LIN {X 0,Y 488.521,Z 455.638,A -85,B 0,C 180,E1 -6694.13,E2 -6694.13} C_VEL
LIN {X 0,Y 488.662,Z 455.615,A -85,B 0,C 180,E1 -6696.351,E2 -6696.351} C_VEL
LIN {X 0,Y 488.705,Z 455.608,A -85,B 0,C 180,E1 -6699.254,E2 -6699.254} C_VEL
LIN {X 0,Y 488.728,Z 455.605,A -85,B 0,C 180,E1 -6701.602,E2 -6701.602} C_VEL
LIN {X 0,Y 488.717,Z 455.607,A -85,B 0,C 180,E1 -6704.802,E2 -6704.802} C_VEL
LIN {X 0,Y 488.696,Z 455.613,A -85,B 0,C 180,E1 -6707.475,E2 -6707.475} C_VEL
LIN {X 0,Y 488.738,Z 455.605,A -85,B 0,C 180,E1 -6709.677,E2 -6709.677} C_VEL
LIN {X 0,Y 488.684,Z 455.611,A -85,B 0,C 180,E1 -6712.841,E2 -6712.841} C_VEL
LIN {X 0,Y 488.736,Z 455.609,A -85,B 0,C 180,E1 -6715.887,E2 -6715.887} C_VEL
LIN {X 0,Y 488.697,Z 455.611,A -85,B 0,C 180,E1 -6718.82,E2 -6718.82} C_VEL
LIN {X 0,Y 488.713,Z 455.608,A -85,B 0,C 180,E1 -6720.348,E2 -6720.348} C_VEL
LIN {X 0,Y 488.06,Z 455.692,A -85,B 0,C 180,E1 -6721.037,E2 -6721.037} C_VEL
LIN {X 0,Y 485.216,Z 456.044,A -85,B 0,C 180,E1 -6722.155,E2 -6722.155} C_VEL
LIN {X 0,Y 482.806,Z 456.345,A -85,B 0,C 180,E1 -6723.056,E2 -6723.056} C_VEL
LIN {X 0,Y 481.776,Z 456.472,A -85,B 0,C 180,E1 -6723.752,E2 -6723.752} C_VEL
LIN {X 0,Y 481.694,Z 456.483,A -85,B 0,C 180,E1 -6723.987,E2 -6723.987} C_VEL
LIN {X 0,Y 481.679,Z 456.482,A -85,B 0,C 180,E1 -6726.812,E2 -6726.812} C_VEL
LIN {X 0,Y 481.701,Z 456.483,A -85,B 0,C 180,E1 -6729.503,E2 -6729.503} C_VEL
LIN {X 0,Y 481.698,Z 456.482,A -85,B 0,C 180,E1 -6732.158,E2 -6732.158} C_VEL
LIN {X 0,Y 481.749,Z 456.478,A -85,B 0,C 180,E1 -6734.776,E2 -6734.776} C_VEL
LIN {X 0,Y 481.757,Z 456.478,A -85,B 0,C 180,E1 -6738.215,E2 -6738.215} C_VEL
LIN {X 0,Y 481.768,Z 456.476,A -85,B 0,C 180,E1 -6741.612,E2 -6741.612} C_VEL
LIN {X 0,Y 481.821,Z 456.467,A -85,B 0,C 180,E1 -6744.14,E2 -6744.14} C_VEL
LIN {X 0,Y 481.933,Z 456.452,A -85,B 0,C 180,E1 -6747.493,E2 -6747.493} C_VEL
LIN {X 0,Y 481.892,Z 456.456,A -85,B 0,C 180,E1 -6750.836,E2 -6750.836} C_VEL
LIN {X 0,Y 481.933,Z 456.452,A -85,B 0,C 180,E1 -6752.507,E2 -6752.507} C_VEL
LIN {X 0,Y 481.804,Z 456.47,A -85,B 0,C 180,E1 -6755.861,E2 -6755.861} C_VEL
LIN {X 0,Y 481.746,Z 456.478,A -85,B 0,C 180,E1 -6758.389,E2 -6758.389} C_VEL
LIN {X 0,Y 481.757,Z 456.475,A -85,B 0,C 180,E1 -6761.785,E2 -6761.785} C_VEL
LIN {X 0,Y 481.749,Z 456.475,A -85,B 0,C 180,E1 -6765.224,E2 -6765.224} C_VEL
LIN {X 0,Y 481.718,Z 456.481,A -85,B 0,C 180,E1 -6768.722,E2 -6768.722} C_VEL
LIN {X 0,Y 481.651,Z 456.488,A -85,B 0,C 180,E1 -6771.395,E2 -6771.395} C_VEL
LIN {X 0,Y 481.667,Z 456.49,A -85,B 0,C 180,E1 -6774.114,E2 -6774.114} C_VEL
LIN {X 0,Y 481.752,Z 456.474,A -85,B 0,C 180,E1 -6777.139,E2 -6777.139} C_VEL
LIN {X 0,Y 481.684,Z 456.485,A -85,B 0,C 180,E1 -6779.741,E2 -6779.741} C_VEL
LIN {X 0,Y 481.677,Z 456.487,A -85,B 0,C 180,E1 -6782.674,E2 -6782.674} C_VEL
LIN {X 0,Y 481.647,Z 456.489,A -85,B 0,C 180,E1 -6785.709,E2 -6785.709} C_VEL
LIN {X 0,Y 481.675,Z 456.482,A -85,B 0,C 180,E1 -6788.859,E2 -6788.859} C_VEL
LIN {X 0,Y 481.657,Z 456.487,A -85,B 0,C 180,E1 -6791.913,E2 -6791.913} C_VEL
LIN {X 0,Y 481.664,Z 456.488,A -85,B 0,C 180,E1 -6794.457,E2 -6794.457} C_VEL
LIN {X 0,Y 481.658,Z 456.488,A -85,B 0,C 180,E1 -6797.84,E2 -6797.84} C_VEL
LIN {X 0,Y 481.684,Z 456.482,A -85,B 0,C 180,E1 -6800.651,E2 -6800.651} C_VEL
LIN {X 0,Y 481.626,Z 456.494,A -85,B 0,C 180,E1 -6803.377,E2 -6803.377} C_VEL
LIN {X 0,Y 481.493,Z 456.51,A -85,B 0,C 180,E1 -6806.312,E2 -6806.312} C_VEL
LIN {X 0,Y 481.114,Z 456.559,A -85,B 0,C 180,E1 -6809.251,E2 -6809.251} C_VEL
LIN {X 0,Y 480.986,Z 456.764,A -85,B 0,C 180,E1 -6810.211,E2 -6810.211} C_VEL
LIN {X 0,Y 481.053,Z 460.075,A -85,B 0,C 180,E1 -6813.07,E2 -6813.07} C_VEL
LIN {X 0,Y 480.958,Z 463.269,A -85,B 0,C 180,E1 -6815.848,E2 -6815.848} C_VEL
LIN {X 0,Y 480.961,Z 467.196,A -85,B 0,C 180,E1 -6819.26,E2 -6819.26} C_VEL
LIN {X 0,Y 480.903,Z 470.487,A -85,B 0,C 180,E1 -6822.127,E2 -6822.127} C_VEL
LIN {X 0,Y 480.927,Z 474.157,A -85,B 0,C 180,E1 -6825.22,E2 -6825.22} C_VEL
LIN {X 0,Y 483.363,Z 485.552,A -85,B 0,C 180,E1 -6825.63,E2 -6825.63} C_VEL
LIN {X 0,Y 483.879,Z 489.967,A -85,B 0,C 180,E1 -6825.812,E2 -6825.812} C_VEL
LIN {X 0,Y 483.545,Z 501.529,A -85,B 0,C 180,E1 -6826.338,E2 -6826.338} C_VEL
LIN {X 0,Y 483.189,Z 513.218,A -85,B 0,C 180,E1 -6827.039,E2 -6827.039} C_VEL
LIN {X 0,Y 482.8,Z 524.711,A -85,B 0,C 180,E1 -6827.921,E2 -6827.921} C_VEL
LIN {X 0,Y 482.34,Z 534.688,A -85,B 0,C 180,E1 -6828.868,E2 -6828.868} C_VEL
LIN {X 0,Y 481.958,Z 543.707,A -85,B 0,C 180,E1 -6829.922,E2 -6829.922} C_VEL
LIN {X 0,Y 481.613,Z 552.483,A -85,B 0,C 180,E1 -6831.186,E2 -6831.186} C_VEL
LIN {X 0,Y 481.294,Z 559.557,A -85,B 0,C 180,E1 -6832.448,E2 -6832.448} C_VEL
LIN {X 0,Y 481.172,Z 565.776,A -85,B 0,C 180,E1 -6833.869,E2 -6833.869} C_VEL
LIN {X 0,Y 481.008,Z 570.825,A -85,B 0,C 180,E1 -6835.39,E2 -6835.39} C_VEL
LIN {X 0,Y 480.913,Z 573.824,A -85,B 0,C 180,E1 -6836.649,E2 -6836.649} C_VEL
LIN {X 0,Y 480.926,Z 575.286,A -85,B 0,C 180,E1 -6837.487,E2 -6837.487} C_VEL
LIN {X 0,Y 480.76,Z 576.965,A -85,B 0,C 180,E1 -6839.162,E2 -6839.162} C_VEL
LIN {X 0,Y 480.745,Z 577.228,A -85,B 0,C 180,E1 -6840,E2 -6840} C_VEL
LIN {X 0,Y 480.76,Z 577.054,A -85,B 0,C 180,E1 -6840.837,E2 -6840.837} C_VEL
LIN {X 0,Y 480.928,Z 575.521,A -85,B 0,C 180,E1 -6842.512,E2 -6842.512} C_VEL
LIN {X 0,Y 480.922,Z 574.16,A -85,B 0,C 180,E1 -6843.351,E2 -6843.351} C_VEL
LIN {X 0,Y 481.007,Z 571.287,A -85,B 0,C 180,E1 -6844.609,E2 -6844.609} C_VEL
LIN {X 0,Y 481.174,Z 566.349,A -85,B 0,C 180,E1 -6846.141,E2 -6846.141} C_VEL
LIN {X 0,Y 481.337,Z 560.311,A -85,B 0,C 180,E1 -6847.551,E2 -6847.551} C_VEL
LIN {X 0,Y 481.621,Z 553.395,A -85,B 0,C 180,E1 -6848.813,E2 -6848.813} C_VEL
LIN {X 0,Y 481.942,Z 544.787,A -85,B 0,C 180,E1 -6850.078,E2 -6850.078} C_VEL
LIN {X 0,Y 482.343,Z 535.961,A -85,B 0,C 180,E1 -6851.131,E2 -6851.131} C_VEL
LIN {X 0,Y 482.771,Z 526.199,A -85,B 0,C 180,E1 -6852.079,E2 -6852.079} C_VEL
LIN {X 0,Y 483.125,Z 514.56,A -85,B 0,C 180,E1 -6852.99,E2 -6852.99} C_VEL
LIN {X 0,Y 483.53,Z 502.682,A -85,B 0,C 180,E1 -6853.715,E2 -6853.715} C_VEL
LIN {X 0,Y 483.91,Z 489.989,A -85,B 0,C 180,E1 -6854.294,E2 -6854.294} C_VEL
LIN {X 0,Y 482.628,Z 482.026,A -85,B 0,C 180,E1 -6854.618,E2 -6854.618} C_VEL
LIN {X 0,Y 481.021,Z 475.218,A -85,B 0,C 180,E1 -6854.868,E2 -6854.868} C_VEL
LIN {X 0,Y 481.048,Z 471.328,A -85,B 0,C 180,E1 -6858.261,E2 -6858.261} C_VEL
LIN {X 0,Y 480.998,Z 467.621,A -85,B 0,C 180,E1 -6861.425,E2 -6861.425} C_VEL
LIN {X 0,Y 481.043,Z 464.368,A -85,B 0,C 180,E1 -6864.147,E2 -6864.147} C_VEL
LIN {X 0,Y 481.084,Z 460.834,A -85,B 0,C 180,E1 -6866.984,E2 -6866.984} C_VEL
LIN {X 0,Y 481.016,Z 456.971,A -85,B 0,C 180,E1 -6869.786,E2 -6869.786} C_VEL
LIN {X 0,Y 481.124,Z 456.558,A -85,B 0,C 180,E1 -6870.748,E2 -6870.748} C_VEL
LIN {X 0,Y 481.507,Z 456.51,A -85,B 0,C 180,E1 -6873.699,E2 -6873.699} C_VEL
LIN {X 0,Y 481.624,Z 456.494,A -85,B 0,C 180,E1 -6876.747,E2 -6876.747} C_VEL
LIN {X 0,Y 481.679,Z 456.486,A -85,B 0,C 180,E1 -6879.94,E2 -6879.94} C_VEL
LIN {X 0,Y 481.669,Z 456.488,A -85,B 0,C 180,E1 -6883.297,E2 -6883.297} C_VEL
LIN {X 0,Y 481.661,Z 456.49,A -85,B 0,C 180,E1 -6885.641,E2 -6885.641} C_VEL
LIN {X 0,Y 481.659,Z 456.489,A -85,B 0,C 180,E1 -6888.958,E2 -6888.958} C_VEL
LIN {X 0,Y 481.719,Z 456.635,A -85,B 0,C 180,E1 -6889.998,E2 -6889.998} C_VEL
LIN {X 0,Y 483.121,Z 464.541,A -85,B 0,C 180,E1 -6893.385,E2 -6893.385} C_VEL
LIN {X 0,Y 483.304,Z 468.523,A -85,B 0,C 180,E1 -6894.987,E2 -6894.987} C_VEL
LIN {X 0,Y 482.858,Z 476.355,A -85,B 0,C 180,E1 -6897.987,E2 -6897.987} C_VEL
LIN {X 0,Y 482.423,Z 484.318,A -85,B 0,C 180,E1 -6900.937,E2 -6900.937} C_VEL
LIN {X 0,Y 482.124,Z 491.72,A -85,B 0,C 180,E1 -6903.602,E2 -6903.602} C_VEL
LIN {X 0,Y 481.857,Z 499.554,A -85,B 0,C 180,E1 -6906.354,E2 -6906.354} C_VEL
LIN {X 0,Y 481.566,Z 508.719,A -85,B 0,C 180,E1 -6909.497,E2 -6909.497} C_VEL
LIN {X 0,Y 481.343,Z 517.918,A -85,B 0,C 180,E1 -6912.583,E2 -6912.583} C_VEL
LIN {X 0,Y 481.207,Z 525.513,A -85,B 0,C 180,E1 -6915.083,E2 -6915.083} C_VEL
LIN {X 0,Y 483.109,Z 538.984,A -85,B 0,C 180,E1 -6915.494,E2 -6915.494} C_VEL
LIN {X 0,Y 483.716,Z 544.262,A -85,B 0,C 180,E1 -6915.7,E2 -6915.7} C_VEL
LIN {X 0,Y 483.348,Z 556.096,A -85,B 0,C 180,E1 -6916.226,E2 -6916.226} C_VEL
LIN {X 0,Y 482.981,Z 567.433,A -85,B 0,C 180,E1 -6916.89,E2 -6916.89} C_VEL
LIN {X 0,Y 482.477,Z 579.715,A -85,B 0,C 180,E1 -6917.809,E2 -6917.809} C_VEL
LIN {X 0,Y 482.083,Z 589.793,A -85,B 0,C 180,E1 -6918.756,E2 -6918.756} C_VEL
LIN {X 0,Y 481.628,Z 599.758,A -85,B 0,C 180,E1 -6919.915,E2 -6919.915} C_VEL
LIN {X 0,Y 481.333,Z 608.553,A -85,B 0,C 180,E1 -6921.181,E2 -6921.181} C_VEL
LIN {X 0,Y 481.107,Z 615.571,A -85,B 0,C 180,E1 -6922.445,E2 -6922.445} C_VEL
LIN {X 0,Y 480.938,Z 621.582,A -85,B 0,C 180,E1 -6923.809,E2 -6923.809} C_VEL
LIN {X 0,Y 480.905,Z 625.601,A -85,B 0,C 180,E1 -6924.97,E2 -6924.97} C_VEL
LIN {X 0,Y 480.858,Z 627.928,A -85,B 0,C 180,E1 -6925.809,E2 -6925.809} C_VEL
LIN {X 0,Y 480.894,Z 629.821,A -85,B 0,C 180,E1 -6926.649,E2 -6926.649} C_VEL
LIN {X 0,Y 480.869,Z 631.238,A -85,B 0,C 180,E1 -6927.487,E2 -6927.487} C_VEL
LIN {X 0,Y 480.824,Z 632.239,A -85,B 0,C 180,E1 -6928.325,E2 -6928.325} C_VEL
LIN {X 0,Y 480.742,Z 633.044,A -85,B 0,C 180,E1 -6930,E2 -6930} C_VEL
LIN {X 0,Y 480.76,Z 632.811,A -85,B 0,C 180,E1 -6930.838,E2 -6930.838} C_VEL
LIN {X 0,Y 480.825,Z 632.176,A -85,B 0,C 180,E1 -6931.675,E2 -6931.675} C_VEL
LIN {X 0,Y 480.881,Z 631.139,A -85,B 0,C 180,E1 -6932.513,E2 -6932.513} C_VEL
LIN {X 0,Y 480.894,Z 629.685,A -85,B 0,C 180,E1 -6933.351,E2 -6933.351} C_VEL
LIN {X 0,Y 480.853,Z 626.643,A -85,B 0,C 180,E1 -6934.611,E2 -6934.611} C_VEL
LIN {X 0,Y 480.953,Z 622.538,A -85,B 0,C 180,E1 -6935.871,E2 -6935.871} C_VEL
LIN {X 0,Y 481.108,Z 616.224,A -85,B 0,C 180,E1 -6937.344,E2 -6937.344} C_VEL
LIN {X 0,Y 481.303,Z 609.329,A -85,B 0,C 180,E1 -6938.608,E2 -6938.608} C_VEL
LIN {X 0,Y 481.537,Z 600.775,A -85,B 0,C 180,E1 -6939.875,E2 -6939.875} C_VEL
LIN {X 0,Y 481.902,Z 591.982,A -85,B 0,C 180,E1 -6940.929,E2 -6940.929} C_VEL
LIN {X 0,Y 482.32,Z 581.32,A -85,B 0,C 180,E1 -6941.972,E2 -6941.972} C_VEL
LIN {X 0,Y 482.723,Z 570.803,A -85,B 0,C 180,E1 -6942.807,E2 -6942.807} C_VEL
LIN {X 0,Y 483.189,Z 558.755,A -85,B 0,C 180,E1 -6943.564,E2 -6943.564} C_VEL
LIN {X 0,Y 483.574,Z 545.487,A -85,B 0,C 180,E1 -6944.197,E2 -6944.197} C_VEL
LIN {X 0,Y 483.219,Z 540.19,A -85,B 0,C 180,E1 -6944.409,E2 -6944.409} C_VEL
LIN {X 0,Y 481.464,Z 526.61,A -85,B 0,C 180,E1 -6944.854,E2 -6944.854} C_VEL
LIN {X 0,Y 481.177,Z 524.25,A -85,B 0,C 180,E1 -6944.918,E2 -6944.918} C_VEL
LIN {X 0,Y 481.251,Z 515.065,A -85,B 0,C 180,E1 -6947.859,E2 -6947.859} C_VEL
LIN {X 0,Y 481.488,Z 505.759,A -85,B 0,C 180,E1 -6950.905,E2 -6950.905} C_VEL
LIN {X 0,Y 481.688,Z 496.306,A -85,B 0,C 180,E1 -6954.113,E2 -6954.113} C_VEL
LIN {X 0,Y 482.022,Z 487.666,A -85,B 0,C 180,E1 -6957.202,E2 -6957.202} C_VEL
LIN {X 0,Y 482.372,Z 479.925,A -85,B 0,C 180,E1 -6960.176,E2 -6960.176} C_VEL
LIN {X 0,Y 482.874,Z 473.051,A -85,B 0,C 180,E1 -6963.079,E2 -6963.079} C_VEL
LIN {X 0,Y 483.32,Z 467.859,A -85,B 0,C 180,E1 -6965.566,E2 -6965.566} C_VEL
LIN {X 0,Y 483.222,Z 465.5,A -85,B 0,C 180,E1 -6966.877,E2 -6966.877} C_VEL
LIN {X 0,Y 482.592,Z 461.645,A -85,B 0,C 180,E1 -6969.48,E2 -6969.48} C_VEL
LIN {X 0,Y 482.074,Z 458.808,A -85,B 0,C 180,E1 -6972.115,E2 -6972.115} C_VEL
LIN {X 0,Y 481.786,Z 457.245,A -85,B 0,C 180,E1 -6974.443,E2 -6974.443} C_VEL
LIN {X 0,Y 481.673,Z 456.489,A -85,B 0,C 180,E1 -6976.848,E2 -6976.848} C_VEL
LIN {X 0,Y 481.679,Z 456.602,A -85,B 0,C 180,E1 -6980.06,E2 -6980.06} C_VEL
LIN {X 0,Y 481.773,Z 457.262,A -85,B 0,C 180,E1 -6982.216,E2 -6982.216} C_VEL
LIN {X 0,Y 481.851,Z 458.489,A -85,B 0,C 180,E1 -6984.764,E2 -6984.764} C_VEL
LIN {X 0,Y 481.721,Z 460.097,A -85,B 0,C 180,E1 -6987.33,E2 -6987.33} C_VEL
LIN {X 0,Y 481.564,Z 462.204,A -85,B 0,C 180,E1 -6990.251,E2 -6990.251} C_VEL
LIN {X 0,Y 481.44,Z 464.478,A -85,B 0,C 180,E1 -6993.094,E2 -6993.094} C_VEL
LIN {X 0,Y 481.289,Z 466.84,A -85,B 0,C 180,E1 -6995.866,E2 -6995.866} C_VEL
LIN {X 0,Y 481.221,Z 470.102,A -85,B 0,C 180,E1 -6999.482,E2 -6999.482} C_VEL
LIN {X 0,Y 481.133,Z 472.621,A -85,B 0,C 180,E1 -7002.137,E2 -7002.137} C_VEL
LIN {X 0,Y 481.11,Z 475.839,A -85,B 0,C 180,E1 -7005.23,E2 -7005.23} C_VEL
LIN {X 0,Y 483.747,Z 487.707,A -85,B 0,C 180,E1 -7005.684,E2 -7005.684} C_VEL
LIN {X 0,Y 483.728,Z 499.221,A -85,B 0,C 180,E1 -7006.183,E2 -7006.183} C_VEL
LIN {X 0,Y 483.295,Z 511.887,A -85,B 0,C 180,E1 -7006.901,E2 -7006.901} C_VEL
LIN {X 0,Y 482.929,Z 522.885,A -85,B 0,C 180,E1 -7007.712,E2 -7007.712} C_VEL
LIN {X 0,Y 482.459,Z 533.264,A -85,B 0,C 180,E1 -7008.659,E2 -7008.659} C_VEL
LIN {X 0,Y 482.094,Z 542.637,A -85,B 0,C 180,E1 -7009.713,E2 -7009.713} C_VEL
LIN {X 0,Y 481.725,Z 551.652,A -85,B 0,C 180,E1 -7010.977,E2 -7010.977} C_VEL
LIN {X 0,Y 481.397,Z 558.919,A -85,B 0,C 180,E1 -7012.239,E2 -7012.239} C_VEL
LIN {X 0,Y 481.213,Z 565.03,A -85,B 0,C 180,E1 -7013.575,E2 -7013.575} C_VEL
LIN {X 0,Y 480.932,Z 569.918,A -85,B 0,C 180,E1 -7014.97,E2 -7014.97} C_VEL
LIN {X 0,Y 481.044,Z 572.203,A -85,B 0,C 180,E1 -7015.811,E2 -7015.811} C_VEL
LIN {X 0,Y 480.922,Z 574.074,A -85,B 0,C 180,E1 -7016.649,E2 -7016.649} C_VEL
LIN {X 0,Y 480.928,Z 575.488,A -85,B 0,C 180,E1 -7017.488,E2 -7017.488} C_VEL
LIN {X 0,Y 480.76,Z 577.088,A -85,B 0,C 180,E1 -7019.163,E2 -7019.163} C_VEL
LIN {X 0,Y 480.744,Z 577.307,A -85,B 0,C 180,E1 -7020,E2 -7020} C_VEL
LIN {X 0,Y 480.76,Z 577.099,A -85,B 0,C 180,E1 -7020.838,E2 -7020.838} C_VEL
LIN {X 0,Y 480.926,Z 575.483,A -85,B 0,C 180,E1 -7022.513,E2 -7022.513} C_VEL
LIN {X 0,Y 480.913,Z 574.091,A -85,B 0,C 180,E1 -7023.351,E2 -7023.351} C_VEL
LIN {X 0,Y 481.003,Z 571.16,A -85,B 0,C 180,E1 -7024.61,E2 -7024.61} C_VEL
LIN {X 0,Y 481.182,Z 566.177,A -85,B 0,C 180,E1 -7026.14,E2 -7026.14} C_VEL
LIN {X 0,Y 481.301,Z 560.075,A -85,B 0,C 180,E1 -7027.552,E2 -7027.552} C_VEL
LIN {X 0,Y 481.599,Z 553.167,A -85,B 0,C 180,E1 -7028.814,E2 -7028.814} C_VEL
LIN {X 0,Y 481.939,Z 544.51,A -85,B 0,C 180,E1 -7030.079,E2 -7030.079} C_VEL
LIN {X 0,Y 482.304,Z 535.641,A -85,B 0,C 180,E1 -7031.133,E2 -7031.133} C_VEL
LIN {X 0,Y 482.769,Z 525.91,A -85,B 0,C 180,E1 -7032.08,E2 -7032.08} C_VEL
LIN {X 0,Y 483.06,Z 515.699,A -85,B 0,C 180,E1 -7032.895,E2 -7032.895} C_VEL
LIN {X 0,Y 483.492,Z 503.394,A -85,B 0,C 180,E1 -7033.663,E2 -7033.663} C_VEL
LIN {X 0,Y 483.857,Z 491.187,A -85,B 0,C 180,E1 -7034.242,E2 -7034.242} C_VEL
LIN {X 0,Y 483.271,Z 484.851,A -85,B 0,C 180,E1 -7034.502,E2 -7034.502} C_VEL
LIN {X 0,Y 480.957,Z 474.164,A -85,B 0,C 180,E1 -7034.898,E2 -7034.898} C_VEL
LIN {X 0,Y 480.962,Z 470.439,A -85,B 0,C 180,E1 -7038.23,E2 -7038.23} C_VEL
LIN {X 0,Y 480.953,Z 466.935,A -85,B 0,C 180,E1 -7041.427,E2 -7041.427} C_VEL
LIN {X 0,Y 480.987,Z 463.983,A -85,B 0,C 180,E1 -7044.15,E2 -7044.15} C_VEL
LIN {X 0,Y 481.089,Z 460.952,A -85,B 0,C 180,E1 -7046.985,E2 -7046.985} C_VEL
LIN {X 0,Y 481.117,Z 457.981,A -85,B 0,C 180,E1 -7049.78,E2 -7049.78} C_VEL
LIN {X 0,Y 481.128,Z 456.962,A -85,B 0,C 180,E1 -7050.748,E2 -7050.748} C_VEL
LIN {X 0,Y 481.22,Z 456.546,A -85,B 0,C 180,E1 -7052.106,E2 -7052.106} C_VEL
LIN {X 0,Y 481.573,Z 456.499,A -85,B 0,C 180,E1 -7055.189,E2 -7055.189} C_VEL
LIN {X 0,Y 481.654,Z 456.487,A -85,B 0,C 180,E1 -7058.007,E2 -7058.007} C_VEL
LIN {X 0,Y 481.667,Z 456.484,A -85,B 0,C 180,E1 -7061.041,E2 -7061.041} C_VEL
LIN {X 0,Y 481.664,Z 456.487,A -85,B 0,C 180,E1 -7064.36,E2 -7064.36} C_VEL
LIN {X 0,Y 481.637,Z 456.491,A -85,B 0,C 180,E1 -7066.853,E2 -7066.853} C_VEL
LIN {X 0,Y 481.681,Z 456.484,A -85,B 0,C 180,E1 -7070.06,E2 -7070.06} C_VEL
LIN {X 0,Y 481.63,Z 456.488,A -85,B 0,C 180,E1 -7073.253,E2 -7073.253} C_VEL
LIN {X 0,Y 481.715,Z 456.48,A -85,B 0,C 180,E1 -7076.33,E2 -7076.33} C_VEL
LIN {X 0,Y 481.656,Z 456.49,A -85,B 0,C 180,E1 -7079.417,E2 -7079.417} C_VEL
LIN {X 0,Y 481.705,Z 456.482,A -85,B 0,C 180,E1 -7082.168,E2 -7082.168} C_VEL
LIN {X 0,Y 481.694,Z 456.483,A -85,B 0,C 180,E1 -7083.987,E2 -7083.987} C_VEL
LIN {X 0,Y 481.031,Z 456.569,A -85,B 0,C 180,E1 -7084.685,E2 -7084.685} C_VEL
LIN {X 0,Y 478.163,Z 456.926,A -85,B 0,C 180,E1 -7085.819,E2 -7085.819} C_VEL
LIN {X 0,Y 475.729,Z 457.226,A -85,B 0,C 180,E1 -7086.732,E2 -7086.732} C_VEL
LIN {X 0,Y 474.677,Z 457.356,A -85,B 0,C 180,E1 -7087.438,E2 -7087.438} C_VEL
LIN {X 0,Y 474.588,Z 457.366,A -85,B 0,C 180,E1 -7087.677,E2 -7087.677} C_VEL
LIN {X 0,Y 474.66,Z 457.36,A -85,B 0,C 180,E1 -7090.09,E2 -7090.09} C_VEL
LIN {X 0,Y 474.645,Z 457.363,A -85,B 0,C 180,E1 -7092.774,E2 -7092.774} C_VEL
LIN {X 0,Y 474.654,Z 457.359,A -85,B 0,C 180,E1 -7095.421,E2 -7095.421} C_VEL
LIN {X 0,Y 474.711,Z 457.356,A -85,B 0,C 180,E1 -7098.038,E2 -7098.038} C_VEL
LIN {X 0,Y 474.733,Z 457.351,A -85,B 0,C 180,E1 -7101.487,E2 -7101.487} C_VEL
LIN {X 0,Y 474.784,Z 457.343,A -85,B 0,C 180,E1 -7104.052,E2 -7104.052} C_VEL
LIN {X 0,Y 474.899,Z 457.329,A -85,B 0,C 180,E1 -7107.455,E2 -7107.455} C_VEL
LIN {X 0,Y 474.918,Z 457.329,A -85,B 0,C 180,E1 -7110,E2 -7110} C_VEL
LIN {X 0,Y 474.899,Z 457.328,A -85,B 0,C 180,E1 -7112.545,E2 -7112.545} C_VEL
LIN {X 0,Y 474.765,Z 457.346,A -85,B 0,C 180,E1 -7115.948,E2 -7115.948} C_VEL
LIN {X 0,Y 474.717,Z 457.355,A -85,B 0,C 180,E1 -7118.514,E2 -7118.514} C_VEL
LIN {X 0,Y 474.711,Z 457.355,A -85,B 0,C 180,E1 -7121.962,E2 -7121.962} C_VEL
LIN {X 0,Y 474.706,Z 457.354,A -85,B 0,C 180,E1 -7125.456,E2 -7125.456} C_VEL
LIN {X 0,Y 474.67,Z 457.359,A -85,B 0,C 180,E1 -7129.01,E2 -7129.01} C_VEL
LIN {X 0,Y 474.594,Z 457.367,A -85,B 0,C 180,E1 -7131.729,E2 -7131.729} C_VEL
LIN {X 0,Y 474.646,Z 457.361,A -85,B 0,C 180,E1 -7134.494,E2 -7134.494} C_VEL
LIN {X 0,Y 474.686,Z 457.355,A -85,B 0,C 180,E1 -7137.334,E2 -7137.334} C_VEL
LIN {X 0,Y 474.61,Z 457.365,A -85,B 0,C 180,E1 -7140.23,E2 -7140.23} C_VEL
LIN {X 0,Y 474.648,Z 457.362,A -85,B 0,C 180,E1 -7143.22,E2 -7143.22} C_VEL
LIN {X 0,Y 474.597,Z 457.368,A -85,B 0,C 180,E1 -7146.323,E2 -7146.323} C_VEL
LIN {X 0,Y 474.632,Z 457.366,A -85,B 0,C 180,E1 -7149.647,E2 -7149.647} C_VEL
LIN {X 0,Y 474.619,Z 457.365,A -85,B 0,C 180,E1 -7152.934,E2 -7152.934} C_VEL
LIN {X 0,Y 474.62,Z 457.364,A -85,B 0,C 180,E1 -7155.896,E2 -7155.896} C_VEL
LIN {X 0,Y 474.637,Z 457.361,A -85,B 0,C 180,E1 -7159.04,E2 -7159.04} C_VEL
LIN {X 0,Y 474.614,Z 457.369,A -85,B 0,C 180,E1 -7161.704,E2 -7161.704} C_VEL
LIN {X 0,Y 474.56,Z 457.372,A -85,B 0,C 180,E1 -7164.72,E2 -7164.72} C_VEL
LIN {X 0,Y 474.296,Z 457.408,A -85,B 0,C 180,E1 -7167.761,E2 -7167.761} C_VEL
LIN {X 0,Y 473.993,Z 457.446,A -85,B 0,C 180,E1 -7169.726,E2 -7169.726} C_VEL
LIN {X 0,Y 473.921,Z 458.298,A -85,B 0,C 180,E1 -7171.038,E2 -7171.038} C_VEL
LIN {X 0,Y 473.947,Z 461.235,A -85,B 0,C 180,E1 -7173.585,E2 -7173.585} C_VEL
LIN {X 0,Y 473.881,Z 465.014,A -85,B 0,C 180,E1 -7176.854,E2 -7176.854} C_VEL
LIN {X 0,Y 473.842,Z 468.655,A -85,B 0,C 180,E1 -7180.054,E2 -7180.054} C_VEL
LIN {X 0,Y 473.8,Z 471.746,A -85,B 0,C 180,E1 -7182.742,E2 -7182.742} C_VEL
LIN {X 0,Y 473.825,Z 474.334,A -85,B 0,C 180,E1 -7184.991,E2 -7184.991} C_VEL
LIN {X 0,Y 476.597,Z 487.342,A -85,B 0,C 180,E1 -7185.482,E2 -7185.482} C_VEL
LIN {X 0,Y 476.931,Z 492.727,A -85,B 0,C 180,E1 -7185.71,E2 -7185.71} C_VEL
LIN {X 0,Y 476.508,Z 505.492,A -85,B 0,C 180,E1 -7186.35,E2 -7186.35} C_VEL
LIN {X 0,Y 476.154,Z 516.762,A -85,B 0,C 180,E1 -7187.087,E2 -7187.087} C_VEL
LIN {X 0,Y 475.767,Z 527.332,A -85,B 0,C 180,E1 -7187.956,E2 -7187.956} C_VEL
LIN {X 0,Y 475.222,Z 536.85,A -85,B 0,C 180,E1 -7188.915,E2 -7188.915} C_VEL
LIN {X 0,Y 474.888,Z 545.56,A -85,B 0,C 180,E1 -7189.986,E2 -7189.986} C_VEL
LIN {X 0,Y 474.52,Z 554.085,A -85,B 0,C 180,E1 -7191.268,E2 -7191.268} C_VEL
LIN {X 0,Y 474.247,Z 560.877,A -85,B 0,C 180,E1 -7192.549,E2 -7192.549} C_VEL
LIN {X 0,Y 474.087,Z 567.112,A -85,B 0,C 180,E1 -7194.043,E2 -7194.043} C_VEL
LIN {X 0,Y 473.926,Z 571.183,A -85,B 0,C 180,E1 -7195.321,E2 -7195.321} C_VEL
LIN {X 0,Y 473.848,Z 574.196,A -85,B 0,C 180,E1 -7196.599,E2 -7196.599} C_VEL
LIN {X 0,Y 473.866,Z 575.667,A -85,B 0,C 180,E1 -7197.45,E2 -7197.45} C_VEL
LIN {X 0,Y 473.689,Z 577.36,A -85,B 0,C 180,E1 -7199.15,E2 -7199.15} C_VEL
LIN {X 0,Y 473.672,Z 577.626,A -85,B 0,C 180,E1 -7200,E2 -7200} C_VEL
LIN {X 0,Y 473.689,Z 577.454,A -85,B 0,C 180,E1 -7200.85,E2 -7200.85} C_VEL
LIN {X 0,Y 473.868,Z 575.922,A -85,B 0,C 180,E1 -7202.55,E2 -7202.55} C_VEL
LIN {X 0,Y 473.856,Z 574.556,A -85,B 0,C 180,E1 -7203.401,E2 -7203.401} C_VEL
LIN {X 0,Y 473.944,Z 571.68,A -85,B 0,C 180,E1 -7204.678,E2 -7204.678} C_VEL
LIN {X 0,Y 474.085,Z 567.755,A -85,B 0,C 180,E1 -7205.956,E2 -7205.956} C_VEL
LIN {X 0,Y 474.218,Z 562.662,A -85,B 0,C 180,E1 -7207.237,E2 -7207.237} C_VEL
LIN {X 0,Y 474.498,Z 556.237,A -85,B 0,C 180,E1 -7208.518,E2 -7208.518} C_VEL
LIN {X 0,Y 474.817,Z 548.257,A -85,B 0,C 180,E1 -7209.8,E2 -7209.8} C_VEL
LIN {X 0,Y 475.204,Z 540.075,A -85,B 0,C 180,E1 -7210.869,E2 -7210.869} C_VEL
LIN {X 0,Y 475.69,Z 529.99,A -85,B 0,C 180,E1 -7211.937,E2 -7211.937} C_VEL
LIN {X 0,Y 476.075,Z 520.102,A -85,B 0,C 180,E1 -7212.793,E2 -7212.793} C_VEL
LIN {X 0,Y 476.455,Z 509.323,A -85,B 0,C 180,E1 -7213.549,E2 -7213.549} C_VEL
LIN {X 0,Y 476.9,Z 497.691,A -85,B 0,C 180,E1 -7214.182,E2 -7214.182} C_VEL
LIN {X 0,Y 476.924,Z 489.024,A -85,B 0,C 180,E1 -7214.561,E2 -7214.561} C_VEL
LIN {X 0,Y 474.354,Z 477.52,A -85,B 0,C 180,E1 -7215.032,E2 -7215.032} C_VEL
LIN {X 0,Y 473.95,Z 475.706,A -85,B 0,C 180,E1 -7215.102,E2 -7215.102} C_VEL
LIN {X 0,Y 473.979,Z 471.927,A -85,B 0,C 180,E1 -7218.382,E2 -7218.382} C_VEL
LIN {X 0,Y 473.934,Z 467.966,A -85,B 0,C 180,E1 -7221.76,E2 -7221.76} C_VEL
LIN {X 0,Y 473.983,Z 464.657,A -85,B 0,C 180,E1 -7224.53,E2 -7224.53} C_VEL
LIN {X 0,Y 474.003,Z 461.036,A -85,B 0,C 180,E1 -7227.363,E2 -7227.363} C_VEL
LIN {X 0,Y 474.009,Z 457.445,A -85,B 0,C 180,E1 -7230.272,E2 -7230.272} C_VEL
LIN {X 0,Y 474.391,Z 457.397,A -85,B 0,C 180,E1 -7233.24,E2 -7233.24} C_VEL
LIN {X 0,Y 474.566,Z 457.373,A -85,B 0,C 180,E1 -7235.46,E2 -7235.46} C_VEL
LIN {X 0,Y 474.613,Z 457.367,A -85,B 0,C 180,E1 -7238.457,E2 -7238.457} C_VEL
LIN {X 0,Y 474.634,Z 457.365,A -85,B 0,C 180,E1 -7240.96,E2 -7240.96} C_VEL
LIN {X 0,Y 474.618,Z 457.366,A -85,B 0,C 180,E1 -7244.104,E2 -7244.104} C_VEL
LIN {X 0,Y 474.617,Z 457.367,A -85,B 0,C 180,E1 -7247.066,E2 -7247.066} C_VEL
LIN {X 0,Y 474.671,Z 457.504,A -85,B 0,C 180,E1 -7249.738,E2 -7249.738} C_VEL
LIN {X 0,Y 475.936,Z 464.709,A -85,B 0,C 180,E1 -7252.883,E2 -7252.883} C_VEL
LIN {X 0,Y 476.32,Z 467.971,A -85,B 0,C 180,E1 -7254.244,E2 -7254.244} C_VEL
LIN {X 0,Y 476.008,Z 474.682,A -85,B 0,C 180,E1 -7256.887,E2 -7256.887} C_VEL
LIN {X 0,Y 475.595,Z 482.436,A -85,B 0,C 180,E1 -7259.839,E2 -7259.839} C_VEL
LIN {X 0,Y 475.216,Z 490.209,A -85,B 0,C 180,E1 -7262.712,E2 -7262.712} C_VEL
LIN {X 0,Y 474.836,Z 499.32,A -85,B 0,C 180,E1 -7265.982,E2 -7265.982} C_VEL
LIN {X 0,Y 474.49,Z 508.457,A -85,B 0,C 180,E1 -7269.177,E2 -7269.177} C_VEL
LIN {X 0,Y 474.3,Z 516.311,A -85,B 0,C 180,E1 -7271.87,E2 -7271.87} C_VEL
LIN {X 0,Y 474.166,Z 525.158,A -85,B 0,C 180,E1 -7274.857,E2 -7274.857} C_VEL
LIN {X 0,Y 476.178,Z 539.625,A -85,B 0,C 180,E1 -7275.319,E2 -7275.319} C_VEL
LIN {X 0,Y 476.792,Z 545.085,A -85,B 0,C 180,E1 -7275.542,E2 -7275.542} C_VEL
LIN {X 0,Y 476.357,Z 557.52,A -85,B 0,C 180,E1 -7276.128,E2 -7276.128} C_VEL
LIN {X 0,Y 475.918,Z 569.57,A -85,B 0,C 180,E1 -7276.877,E2 -7276.877} C_VEL
LIN {X 0,Y 475.419,Z 580.793,A -85,B 0,C 180,E1 -7277.765,E2 -7277.765} C_VEL
LIN {X 0,Y 475.031,Z 590.292,A -85,B 0,C 180,E1 -7278.695,E2 -7278.695} C_VEL
LIN {X 0,Y 474.593,Z 599.29,A -85,B 0,C 180,E1 -7279.764,E2 -7279.764} C_VEL
LIN {X 0,Y 474.272,Z 608.103,A -85,B 0,C 180,E1 -7281.049,E2 -7281.049} C_VEL
LIN {X 0,Y 474.038,Z 615.137,A -85,B 0,C 180,E1 -7282.332,E2 -7282.332} C_VEL
LIN {X 0,Y 473.88,Z 620.512,A -85,B 0,C 180,E1 -7283.547,E2 -7283.547} C_VEL
LIN {X 0,Y 473.839,Z 625.188,A -85,B 0,C 180,E1 -7284.894,E2 -7284.894} C_VEL
LIN {X 0,Y 473.76,Z 627.516,A -85,B 0,C 180,E1 -7285.746,E2 -7285.746} C_VEL
LIN {X 0,Y 473.82,Z 629.414,A -85,B 0,C 180,E1 -7286.599,E2 -7286.599} C_VEL
LIN {X 0,Y 473.783,Z 630.833,A -85,B 0,C 180,E1 -7287.449,E2 -7287.449} C_VEL
LIN {X 0,Y 473.758,Z 631.834,A -85,B 0,C 180,E1 -7288.3,E2 -7288.3} C_VEL
LIN {X 0,Y 473.688,Z 632.434,A -85,B 0,C 180,E1 -7289.15,E2 -7289.15} C_VEL
LIN {X 0,Y 473.669,Z 632.636,A -85,B 0,C 180,E1 -7290,E2 -7290} C_VEL
LIN {X 0,Y 473.688,Z 632.399,A -85,B 0,C 180,E1 -7290.85,E2 -7290.85} C_VEL
LIN {X 0,Y 473.758,Z 631.756,A -85,B 0,C 180,E1 -7291.7,E2 -7291.7} C_VEL
LIN {X 0,Y 473.793,Z 630.71,A -85,B 0,C 180,E1 -7292.551,E2 -7292.551} C_VEL
LIN {X 0,Y 473.821,Z 629.249,A -85,B 0,C 180,E1 -7293.401,E2 -7293.401} C_VEL
LIN {X 0,Y 473.775,Z 626.189,A -85,B 0,C 180,E1 -7294.68,E2 -7294.68} C_VEL
LIN {X 0,Y 473.859,Z 622.061,A -85,B 0,C 180,E1 -7295.959,E2 -7295.959} C_VEL
LIN {X 0,Y 474.017,Z 615.71,A -85,B 0,C 180,E1 -7297.454,E2 -7297.454} C_VEL
LIN {X 0,Y 474.213,Z 608.786,A -85,B 0,C 180,E1 -7298.738,E2 -7298.738} C_VEL
LIN {X 0,Y 474.495,Z 600.204,A -85,B 0,C 180,E1 -7300.023,E2 -7300.023} C_VEL
LIN {X 0,Y 474.897,Z 591.382,A -85,B 0,C 180,E1 -7301.092,E2 -7301.092} C_VEL
LIN {X 0,Y 475.329,Z 580.969,A -85,B 0,C 180,E1 -7302.126,E2 -7302.126} C_VEL
LIN {X 0,Y 475.791,Z 569.875,A -85,B 0,C 180,E1 -7303.018,E2 -7303.018} C_VEL
LIN {X 0,Y 476.238,Z 558.098,A -85,B 0,C 180,E1 -7303.766,E2 -7303.766} C_VEL
LIN {X 0,Y 476.671,Z 544.885,A -85,B 0,C 180,E1 -7304.407,E2 -7304.407} C_VEL
LIN {X 0,Y 475.105,Z 531.598,A -85,B 0,C 180,E1 -7304.921,E2 -7304.921} C_VEL
LIN {X 0,Y 474.114,Z 523.769,A -85,B 0,C 180,E1 -7305.145,E2 -7305.145} C_VEL
LIN {X 0,Y 474.241,Z 513.587,A -85,B 0,C 180,E1 -7308.477,E2 -7308.477} C_VEL
LIN {X 0,Y 474.465,Z 503.913,A -85,B 0,C 180,E1 -7311.735,E2 -7311.735} C_VEL
LIN {X 0,Y 474.736,Z 494.736,A -85,B 0,C 180,E1 -7314.956,E2 -7314.956} C_VEL
LIN {X 0,Y 475.041,Z 487.111,A -85,B 0,C 180,E1 -7317.786,E2 -7317.786} C_VEL
LIN {X 0,Y 475.545,Z 478.74,A -85,B 0,C 180,E1 -7321.149,E2 -7321.149} C_VEL
LIN {X 0,Y 476.132,Z 471.877,A -85,B 0,C 180,E1 -7324.249,E2 -7324.249} C_VEL
LIN {X 0,Y 476.319,Z 468.198,A -85,B 0,C 180,E1 -7326.171,E2 -7326.171} C_VEL
LIN {X 0,Y 475.912,Z 464.512,A -85,B 0,C 180,E1 -7328.494,E2 -7328.494} C_VEL
LIN {X 0,Y 475.366,Z 461.397,A -85,B 0,C 180,E1 -7331.061,E2 -7331.061} C_VEL
LIN {X 0,Y 474.94,Z 459.349,A -85,B 0,C 180,E1 -7333.524,E2 -7333.524} C_VEL
LIN {X 0,Y 474.745,Z 458.223,A -85,B 0,C 180,E1 -7335.911,E2 -7335.911} C_VEL
LIN {X 0,Y 474.711,Z 457.857,A -85,B 0,C 180,E1 -7338.224,E2 -7338.224} C_VEL
LIN {X 0,Y 474.718,Z 458.081,A -85,B 0,C 180,E1 -7340.461,E2 -7340.461} C_VEL
LIN {X 0,Y 474.805,Z 458.912,A -85,B 0,C 180,E1 -7343.064,E2 -7343.064} C_VEL
LIN {X 0,Y 474.789,Z 460.268,A -85,B 0,C 180,E1 -7345.772,E2 -7345.772} C_VEL
LIN {X 0,Y 474.628,Z 462.195,A -85,B 0,C 180,E1 -7348.785,E2 -7348.785} C_VEL
LIN {X 0,Y 474.456,Z 464.361,A -85,B 0,C 180,E1 -7351.705,E2 -7351.705} C_VEL
LIN {X 0,Y 474.315,Z 466.748,A -85,B 0,C 180,E1 -7354.669,E2 -7354.669} C_VEL
LIN {X 0,Y 474.176,Z 469.041,A -85,B 0,C 180,E1 -7357.334,E2 -7357.334} C_VEL
LIN {X 0,Y 474.091,Z 471.502,A -85,B 0,C 180,E1 -7360.065,E2 -7360.065} C_VEL
LIN {X 0,Y 474.043,Z 474.028,A -85,B 0,C 180,E1 -7362.752,E2 -7362.752} C_VEL
LIN {X 0,Y 474.039,Z 476.2,A -85,B 0,C 180,E1 -7364.985,E2 -7364.985} C_VEL
LIN {X 0,Y 476.869,Z 488.579,A -85,B 0,C 180,E1 -7365.49,E2 -7365.49} C_VEL
LIN {X 0,Y 476.863,Z 499.583,A -85,B 0,C 180,E1 -7365.98,E2 -7365.98} C_VEL
LIN {X 0,Y 476.481,Z 511.092,A -85,B 0,C 180,E1 -7366.634,E2 -7366.634} C_VEL
LIN {X 0,Y 476.058,Z 521.991,A -85,B 0,C 180,E1 -7367.423,E2 -7367.423} C_VEL
LIN {X 0,Y 475.575,Z 532.592,A -85,B 0,C 180,E1 -7368.384,E2 -7368.384} C_VEL
LIN {X 0,Y 475.183,Z 541.279,A -85,B 0,C 180,E1 -7369.346,E2 -7369.346} C_VEL
LIN {X 0,Y 474.849,Z 549.269,A -85,B 0,C 180,E1 -7370.415,E2 -7370.415} C_VEL
LIN {X 0,Y 474.475,Z 557.108,A -85,B 0,C 180,E1 -7371.697,E2 -7371.697} C_VEL
LIN {X 0,Y 474.248,Z 562.398,A -85,B 0,C 180,E1 -7372.764,E2 -7372.764} C_VEL
LIN {X 0,Y 474.102,Z 567.557,A -85,B 0,C 180,E1 -7374.044,E2 -7374.044} C_VEL
LIN {X 0,Y 473.947,Z 571.551,A -85,B 0,C 180,E1 -7375.322,E2 -7375.322} C_VEL
LIN {X 0,Y 473.856,Z 574.488,A -85,B 0,C 180,E1 -7376.599,E2 -7376.599} C_VEL
LIN {X 0,Y 473.868,Z 575.904,A -85,B 0,C 180,E1 -7377.45,E2 -7377.45} C_VEL
LIN {X 0,Y 473.689,Z 577.502,A -85,B 0,C 180,E1 -7379.15,E2 -7379.15} C_VEL
LIN {X 0,Y 473.671,Z 577.718,A -85,B 0,C 180,E1 -7380,E2 -7380} C_VEL
LIN {X 0,Y 473.689,Z 577.507,A -85,B 0,C 180,E1 -7380.85,E2 -7380.85} C_VEL
LIN {X 0,Y 473.866,Z 575.875,A -85,B 0,C 180,E1 -7382.55,E2 -7382.55} C_VEL
LIN {X 0,Y 473.848,Z 574.476,A -85,B 0,C 180,E1 -7383.401,E2 -7383.401} C_VEL
LIN {X 0,Y 473.939,Z 571.53,A -85,B 0,C 180,E1 -7384.678,E2 -7384.678} C_VEL
LIN {X 0,Y 474.09,Z 567.545,A -85,B 0,C 180,E1 -7385.957,E2 -7385.957} C_VEL
LIN {X 0,Y 474.257,Z 561.411,A -85,B 0,C 180,E1 -7387.451,E2 -7387.451} C_VEL
LIN {X 0,Y 474.51,Z 554.704,A -85,B 0,C 180,E1 -7388.732,E2 -7388.732} C_VEL
LIN {X 0,Y 474.867,Z 546.385,A -85,B 0,C 180,E1 -7390.015,E2 -7390.015} C_VEL
LIN {X 0,Y 475.197,Z 537.831,A -85,B 0,C 180,E1 -7391.085,E2 -7391.085} C_VEL
LIN {X 0,Y 475.782,Z 527.293,A -85,B 0,C 180,E1 -7392.152,E2 -7392.152} C_VEL
LIN {X 0,Y 476.125,Z 516.51,A -85,B 0,C 180,E1 -7393.038,E2 -7393.038} C_VEL
LIN {X 0,Y 476.534,Z 505.489,A -85,B 0,C 180,E1 -7393.758,E2 -7393.758} C_VEL
LIN {X 0,Y 476.946,Z 492.57,A -85,B 0,C 180,E1 -7394.399,E2 -7394.399} C_VEL
LIN {X 0,Y 476.547,Z 486.903,A -85,B 0,C 180,E1 -7394.638,E2 -7394.638} C_VEL
LIN {X 0,Y 473.91,Z 474.484,A -85,B 0,C 180,E1 -7395.115,E2 -7395.115} C_VEL
LIN {X 0,Y 473.905,Z 470.893,A -85,B 0,C 180,E1 -7398.355,E2 -7398.355} C_VEL
LIN {X 0,Y 473.882,Z 467.171,A -85,B 0,C 180,E1 -7401.763,E2 -7401.763} C_VEL
LIN {X 0,Y 473.925,Z 464.191,A -85,B 0,C 180,E1 -7404.534,E2 -7404.534} C_VEL
LIN {X 0,Y 474.021,Z 461.181,A -85,B 0,C 180,E1 -7407.363,E2 -7407.363} C_VEL
LIN {X 0,Y 474.061,Z 457.675,A -85,B 0,C 180,E1 -7410.699,E2 -7410.699} C_VEL
LIN {X 0,Y 474.312,Z 457.405,A -85,B 0,C 180,E1 -7413.247,E2 -7413.247} C_VEL
LIN {X 0,Y 474.55,Z 457.374,A -85,B 0,C 180,E1 -7415.458,E2 -7415.458} C_VEL
LIN {X 0,Y 474.614,Z 457.367,A -85,B 0,C 180,E1 -7418.458,E2 -7418.458} C_VEL
LIN {X 0,Y 474.633,Z 457.362,A -85,B 0,C 180,E1 -7421.785,E2 -7421.785} C_VEL
LIN {X 0,Y 474.626,Z 457.362,A -85,B 0,C 180,E1 -7424.703,E2 -7424.703} C_VEL
LIN {X 0,Y 474.625,Z 457.363,A -85,B 0,C 180,E1 -7428.215,E2 -7428.215} C_VEL
LIN {X 0,Y 474.649,Z 457.363,A -85,B 0,C 180,E1 -7430.454,E2 -7430.454} C_VEL
LIN {X 0,Y 474.594,Z 457.366,A -85,B 0,C 180,E1 -7433.677,E2 -7433.677} C_VEL
LIN {X 0,Y 474.648,Z 457.36,A -85,B 0,C 180,E1 -7436.78,E2 -7436.78} C_VEL
LIN {X 0,Y 474.611,Z 457.366,A -85,B 0,C 180,E1 -7439.77,E2 -7439.77} C_VEL
LIN {X 0,Y 474.702,Z 457.356,A -85,B 0,C 180,E1 -7442.68,E2 -7442.68} C_VEL
LIN {X 0,Y 474.646,Z 457.359,A -85,B 0,C 180,E1 -7445.506,E2 -7445.506} C_VEL
LIN {X 0,Y 474.588,Z 457.366,A -85,B 0,C 180,E1 -7447.677,E2 -7447.677} C_VEL
LIN {X 0,Y 473.916,Z 457.452,A -85,B 0,C 180,E1 -7448.385,E2 -7448.385} C_VEL
LIN {X 0,Y 471.08,Z 457.806,A -85,B 0,C 180,E1 -7449.537,E2 -7449.537} C_VEL
LIN {X 0,Y 468.7,Z 458.102,A -85,B 0,C 180,E1 -7450.465,E2 -7450.465} C_VEL
LIN {X 0,Y 467.695,Z 458.228,A -85,B 0,C 180,E1 -7451.182,E2 -7451.182} C_VEL
LIN {X 0,Y 467.622,Z 458.237,A -85,B 0,C 180,E1 -7451.424,E2 -7451.424} C_VEL
LIN {X 0,Y 467.645,Z 458.234,A -85,B 0,C 180,E1 -7454.305,E2 -7454.305} C_VEL
LIN {X 0,Y 467.662,Z 458.231,A -85,B 0,C 180,E1 -7457.855,E2 -7457.855} C_VEL
LIN {X 0,Y 467.686,Z 458.228,A -85,B 0,C 180,E1 -7461.357,E2 -7461.357} C_VEL
LIN {X 0,Y 467.749,Z 458.22,A -85,B 0,C 180,E1 -7463.963,E2 -7463.963} C_VEL
LIN {X 0,Y 467.865,Z 458.205,A -85,B 0,C 180,E1 -7467.417,E2 -7467.417} C_VEL
LIN {X 0,Y 467.888,Z 458.205,A -85,B 0,C 180,E1 -7470,E2 -7470} C_VEL
LIN {X 0,Y 467.865,Z 458.204,A -85,B 0,C 180,E1 -7472.583,E2 -7472.583} C_VEL
LIN {X 0,Y 467.727,Z 458.223,A -85,B 0,C 180,E1 -7476.038,E2 -7476.038} C_VEL
LIN {X 0,Y 467.675,Z 458.231,A -85,B 0,C 180,E1 -7478.643,E2 -7478.643} C_VEL
LIN {X 0,Y 467.662,Z 458.234,A -85,B 0,C 180,E1 -7482.145,E2 -7482.145} C_VEL
LIN {X 0,Y 467.645,Z 458.236,A -85,B 0,C 180,E1 -7485.695,E2 -7485.695} C_VEL
LIN {X 0,Y 467.623,Z 458.237,A -85,B 0,C 180,E1 -7488.764,E2 -7488.764} C_VEL
LIN {X 0,Y 467.586,Z 458.241,A -85,B 0,C 180,E1 -7491.268,E2 -7491.268} C_VEL
LIN {X 0,Y 467.569,Z 458.245,A -85,B 0,C 180,E1 -7493.944,E2 -7493.944} C_VEL
LIN {X 0,Y 467.618,Z 458.233,A -85,B 0,C 180,E1 -7496.8,E2 -7496.8} C_VEL
LIN {X 0,Y 467.559,Z 458.245,A -85,B 0,C 180,E1 -7499.738,E2 -7499.738} C_VEL
LIN {X 0,Y 467.588,Z 458.241,A -85,B 0,C 180,E1 -7502.758,E2 -7502.758} C_VEL
LIN {X 0,Y 467.561,Z 458.245,A -85,B 0,C 180,E1 -7505.889,E2 -7505.889} C_VEL
LIN {X 0,Y 467.587,Z 458.238,A -85,B 0,C 180,E1 -7509.145,E2 -7509.145} C_VEL
LIN {X 0,Y 467.591,Z 458.24,A -85,B 0,C 180,E1 -7512.567,E2 -7512.567} C_VEL
LIN {X 0,Y 467.575,Z 458.243,A -85,B 0,C 180,E1 -7515.053,E2 -7515.053} C_VEL
LIN {X 0,Y 467.593,Z 458.239,A -85,B 0,C 180,E1 -7517.44,E2 -7517.44} C_VEL
LIN {X 0,Y 467.586,Z 458.238,A -85,B 0,C 180,E1 -7520.855,E2 -7520.855} C_VEL
LIN {X 0,Y 467.511,Z 458.249,A -85,B 0,C 180,E1 -7524.106,E2 -7524.106} C_VEL
LIN {X 0,Y 467.408,Z 458.265,A -85,B 0,C 180,E1 -7526.197,E2 -7526.197} C_VEL
LIN {X 0,Y 467.03,Z 458.313,A -85,B 0,C 180,E1 -7529.226,E2 -7529.226} C_VEL
LIN {X 0,Y 466.857,Z 458.666,A -85,B 0,C 180,E1 -7530.824,E2 -7530.824} C_VEL
LIN {X 0,Y 466.897,Z 461.326,A -85,B 0,C 180,E1 -7533.155,E2 -7533.155} C_VEL
LIN {X 0,Y 466.786,Z 464.61,A -85,B 0,C 180,E1 -7536.013,E2 -7536.013} C_VEL
LIN {X 0,Y 466.794,Z 468.024,A -85,B 0,C 180,E1 -7538.982,E2 -7538.982} C_VEL
LIN {X 0,Y 466.755,Z 470.963,A -85,B 0,C 180,E1 -7541.566,E2 -7541.566} C_VEL
LIN {X 0,Y 466.743,Z 474.716,A -85,B 0,C 180,E1 -7544.782,E2 -7544.782} C_VEL
LIN {X 0,Y 469.497,Z 487.221,A -85,B 0,C 180,E1 -7545.257,E2 -7545.257} C_VEL
LIN {X 0,Y 470.059,Z 492.675,A -85,B 0,C 180,E1 -7545.496,E2 -7545.496} C_VEL
LIN {X 0,Y 469.599,Z 505.522,A -85,B 0,C 180,E1 -7546.145,E2 -7546.145} C_VEL
LIN {X 0,Y 469.209,Z 517.581,A -85,B 0,C 180,E1 -7546.947,E2 -7546.947} C_VEL
LIN {X 0,Y 468.753,Z 528.615,A -85,B 0,C 180,E1 -7547.883,E2 -7547.883} C_VEL
LIN {X 0,Y 468.195,Z 538.937,A -85,B 0,C 180,E1 -7548.966,E2 -7548.966} C_VEL
LIN {X 0,Y 467.811,Z 547.374,A -85,B 0,C 180,E1 -7550.051,E2 -7550.051} C_VEL
LIN {X 0,Y 467.438,Z 555.57,A -85,B 0,C 180,E1 -7551.352,E2 -7551.352} C_VEL
LIN {X 0,Y 467.168,Z 562.173,A -85,B 0,C 180,E1 -7552.653,E2 -7552.653} C_VEL
LIN {X 0,Y 467.04,Z 567.436,A -85,B 0,C 180,E1 -7553.953,E2 -7553.953} C_VEL
LIN {X 0,Y 466.852,Z 571.531,A -85,B 0,C 180,E1 -7555.25,E2 -7555.25} C_VEL
LIN {X 0,Y 466.786,Z 574.561,A -85,B 0,C 180,E1 -7556.547,E2 -7556.547} C_VEL
LIN {X 0,Y 466.777,Z 576.046,A -85,B 0,C 180,E1 -7557.411,E2 -7557.411} C_VEL
LIN {X 0,Y 466.62,Z 577.752,A -85,B 0,C 180,E1 -7559.137,E2 -7559.137} C_VEL
LIN {X 0,Y 466.6,Z 578.026,A -85,B 0,C 180,E1 -7560,E2 -7560} C_VEL
LIN {X 0,Y 466.62,Z 577.859,A -85,B 0,C 180,E1 -7560.863,E2 -7560.863} C_VEL
LIN {X 0,Y 466.809,Z 576.333,A -85,B 0,C 180,E1 -7562.589,E2 -7562.589} C_VEL
LIN {X 0,Y 466.793,Z 574.97,A -85,B 0,C 180,E1 -7563.452,E2 -7563.452} C_VEL
LIN {X 0,Y 466.883,Z 572.093,A -85,B 0,C 180,E1 -7564.749,E2 -7564.749} C_VEL
LIN {X 0,Y 467.042,Z 568.163,A -85,B 0,C 180,E1 -7566.046,E2 -7566.046} C_VEL
LIN {X 0,Y 467.198,Z 563.061,A -85,B 0,C 180,E1 -7567.346,E2 -7567.346} C_VEL
LIN {X 0,Y 467.474,Z 556.626,A -85,B 0,C 180,E1 -7568.646,E2 -7568.646} C_VEL
LIN {X 0,Y 467.846,Z 548.631,A -85,B 0,C 180,E1 -7569.948,E2 -7569.948} C_VEL
LIN {X 0,Y 468.244,Z 540.429,A -85,B 0,C 180,E1 -7571.033,E2 -7571.033} C_VEL
LIN {X 0,Y 468.815,Z 529.235,A -85,B 0,C 180,E1 -7572.225,E2 -7572.225} C_VEL
LIN {X 0,Y 469.243,Z 518.988,A -85,B 0,C 180,E1 -7573.106,E2 -7573.106} C_VEL
LIN {X 0,Y 469.656,Z 508.133,A -85,B 0,C 180,E1 -7573.853,E2 -7573.853} C_VEL
LIN {X 0,Y 470.138,Z 494.832,A -85,B 0,C 180,E1 -7574.556,E2 -7574.556} C_VEL
LIN {X 0,Y 470.048,Z 489.928,A -85,B 0,C 180,E1 -7574.77,E2 -7574.77} C_VEL
LIN {X 0,Y 467.429,Z 478.311,A -85,B 0,C 180,E1 -7575.265,E2 -7575.265} C_VEL
LIN {X 0,Y 466.914,Z 476.176,A -85,B 0,C 180,E1 -7575.352,E2 -7575.352} C_VEL
LIN {X 0,Y 466.916,Z 472.559,A -85,B 0,C 180,E1 -7578.508,E2 -7578.508} C_VEL
LIN {X 0,Y 466.892,Z 469.457,A -85,B 0,C 180,E1 -7581.178,E2 -7581.178} C_VEL
LIN {X 0,Y 466.911,Z 466.113,A -85,B 0,C 180,E1 -7583.979,E2 -7583.979} C_VEL
LIN {X 0,Y 466.959,Z 463.798,A -85,B 0,C 180,E1 -7585.879,E2 -7585.879} C_VEL
LIN {X 0,Y 466.936,Z 461.352,A -85,B 0,C 180,E1 -7587.813,E2 -7587.813} C_VEL
LIN {X 0,Y 466.899,Z 458.674,A -85,B 0,C 180,E1 -7589.784,E2 -7589.784} C_VEL
LIN {X 0,Y 467.174,Z 458.296,A -85,B 0,C 180,E1 -7591.771,E2 -7591.771} C_VEL
LIN {X 0,Y 467.479,Z 458.256,A -85,B 0,C 180,E1 -7594.84,E2 -7594.84} C_VEL
LIN {X 0,Y 467.567,Z 458.245,A -85,B 0,C 180,E1 -7598.044,E2 -7598.044} C_VEL
LIN {X 0,Y 467.584,Z 458.242,A -85,B 0,C 180,E1 -7601.277,E2 -7601.277} C_VEL
LIN {X 0,Y 467.569,Z 458.244,A -85,B 0,C 180,E1 -7603.823,E2 -7603.823} C_VEL
LIN {X 0,Y 467.558,Z 458.246,A -85,B 0,C 180,E1 -7606.256,E2 -7606.256} C_VEL
LIN {X 0,Y 467.613,Z 458.343,A -85,B 0,C 180,E1 -7609.456,E2 -7609.456} C_VEL
LIN {X 0,Y 468.869,Z 465.41,A -85,B 0,C 180,E1 -7612.602,E2 -7612.602} C_VEL
LIN {X 0,Y 469.356,Z 469.337,A -85,B 0,C 180,E1 -7614.269,E2 -7614.269} C_VEL
LIN {X 0,Y 468.979,Z 476.323,A -85,B 0,C 180,E1 -7617.056,E2 -7617.056} C_VEL
LIN {X 0,Y 468.578,Z 483.516,A -85,B 0,C 180,E1 -7619.837,E2 -7619.837} C_VEL
LIN {X 0,Y 468.157,Z 491.35,A -85,B 0,C 180,E1 -7622.774,E2 -7622.774} C_VEL
LIN {X 0,Y 467.773,Z 500.374,A -85,B 0,C 180,E1 -7626.068,E2 -7626.068} C_VEL
LIN {X 0,Y 467.423,Z 509.493,A -85,B 0,C 180,E1 -7629.308,E2 -7629.308} C_VEL
LIN {X 0,Y 467.215,Z 517.321,A -85,B 0,C 180,E1 -7632.039,E2 -7632.039} C_VEL
LIN {X 0,Y 467.098,Z 524.821,A -85,B 0,C 180,E1 -7634.619,E2 -7634.619} C_VEL
LIN {X 0,Y 469.207,Z 540.251,A -85,B 0,C 180,E1 -7635.142,E2 -7635.142} C_VEL
LIN {X 0,Y 469.836,Z 545.775,A -85,B 0,C 180,E1 -7635.379,E2 -7635.379} C_VEL
LIN {X 0,Y 469.359,Z 558.91,A -85,B 0,C 180,E1 -7636.028,E2 -7636.028} C_VEL
LIN {X 0,Y 468.893,Z 570.55,A -85,B 0,C 180,E1 -7636.787,E2 -7636.787} C_VEL
LIN {X 0,Y 468.376,Z 581.575,A -85,B 0,C 180,E1 -7637.698,E2 -7637.698} C_VEL
LIN {X 0,Y 467.927,Z 591.765,A -85,B 0,C 180,E1 -7638.74,E2 -7638.74} C_VEL
LIN {X 0,Y 467.485,Z 600.458,A -85,B 0,C 180,E1 -7639.826,E2 -7639.826} C_VEL
LIN {X 0,Y 467.163,Z 608.913,A -85,B 0,C 180,E1 -7641.129,E2 -7641.129} C_VEL
LIN {X 0,Y 466.928,Z 615.722,A -85,B 0,C 180,E1 -7642.432,E2 -7642.432} C_VEL
LIN {X 0,Y 466.768,Z 621.972,A -85,B 0,C 180,E1 -7643.95,E2 -7643.95} C_VEL
LIN {X 0,Y 466.701,Z 626.021,A -85,B 0,C 180,E1 -7645.249,E2 -7645.249} C_VEL
LIN {X 0,Y 466.73,Z 629.006,A -85,B 0,C 180,E1 -7646.547,E2 -7646.547} C_VEL
LIN {X 0,Y 466.7,Z 630.428,A -85,B 0,C 180,E1 -7647.411,E2 -7647.411} C_VEL
LIN {X 0,Y 466.693,Z 631.429,A -85,B 0,C 180,E1 -7648.274,E2 -7648.274} C_VEL
LIN {X 0,Y 466.62,Z 632.028,A -85,B 0,C 180,E1 -7649.137,E2 -7649.137} C_VEL
LIN {X 0,Y 466.598,Z 632.228,A -85,B 0,C 180,E1 -7650,E2 -7650} C_VEL
LIN {X 0,Y 466.62,Z 631.984,A -85,B 0,C 180,E1 -7650.863,E2 -7650.863} C_VEL
LIN {X 0,Y 466.694,Z 631.335,A -85,B 0,C 180,E1 -7651.726,E2 -7651.726} C_VEL
LIN {X 0,Y 466.71,Z 630.282,A -85,B 0,C 180,E1 -7652.589,E2 -7652.589} C_VEL
LIN {X 0,Y 466.73,Z 628.811,A -85,B 0,C 180,E1 -7653.453,E2 -7653.453} C_VEL
LIN {X 0,Y 466.701,Z 625.736,A -85,B 0,C 180,E1 -7654.751,E2 -7654.751} C_VEL
LIN {X 0,Y 466.773,Z 621.588,A -85,B 0,C 180,E1 -7656.05,E2 -7656.05} C_VEL
LIN {X 0,Y 466.928,Z 615.211,A -85,B 0,C 180,E1 -7657.568,E2 -7657.568} C_VEL
LIN {X 0,Y 467.142,Z 608.265,A -85,B 0,C 180,E1 -7658.871,E2 -7658.871} C_VEL
LIN {X 0,Y 467.463,Z 599.65,A -85,B 0,C 180,E1 -7660.175,E2 -7660.175} C_VEL
LIN {X 0,Y 467.909,Z 590.817,A -85,B 0,C 180,E1 -7661.26,E2 -7661.26} C_VEL
LIN {X 0,Y 468.338,Z 580.645,A -85,B 0,C 180,E1 -7662.287,E2 -7662.287} C_VEL
LIN {X 0,Y 468.818,Z 569.321,A -85,B 0,C 180,E1 -7663.215,E2 -7663.215} C_VEL
LIN {X 0,Y 469.3,Z 557.558,A -85,B 0,C 180,E1 -7663.974,E2 -7663.974} C_VEL
LIN {X 0,Y 469.698,Z 544.432,A -85,B 0,C 180,E1 -7664.625,E2 -7664.625} C_VEL
LIN {X 0,Y 468.068,Z 531.191,A -85,B 0,C 180,E1 -7665.157,E2 -7665.157} C_VEL
LIN {X 0,Y 467.019,Z 523.224,A -85,B 0,C 180,E1 -7665.409,E2 -7665.409} C_VEL
LIN {X 0,Y 467.168,Z 513.678,A -85,B 0,C 180,E1 -7668.601,E2 -7668.601} C_VEL
LIN {X 0,Y 467.391,Z 504.9,A -85,B 0,C 180,E1 -7671.617,E2 -7671.617} C_VEL
LIN {X 0,Y 467.664,Z 495.775,A -85,B 0,C 180,E1 -7674.884,E2 -7674.884} C_VEL
LIN {X 0,Y 468.02,Z 488.237,A -85,B 0,C 180,E1 -7677.743,E2 -7677.743} C_VEL
LIN {X 0,Y 468.558,Z 479.713,A -85,B 0,C 180,E1 -7681.245,E2 -7681.245} C_VEL
LIN {X 0,Y 469.038,Z 474.433,A -85,B 0,C 180,E1 -7683.67,E2 -7683.67} C_VEL
LIN {X 0,Y 469.374,Z 469.86,A -85,B 0,C 180,E1 -7686.045,E2 -7686.045} C_VEL
LIN {X 0,Y 469.096,Z 466.887,A -85,B 0,C 180,E1 -7687.899,E2 -7687.899} C_VEL
LIN {X 0,Y 468.574,Z 463.943,A -85,B 0,C 180,E1 -7690.162,E2 -7690.162} C_VEL
LIN {X 0,Y 468.164,Z 461.563,A -85,B 0,C 180,E1 -7692.644,E2 -7692.644} C_VEL
LIN {X 0,Y 467.905,Z 460.072,A -85,B 0,C 180,E1 -7695.094,E2 -7695.094} C_VEL
LIN {X 0,Y 467.786,Z 459.398,A -85,B 0,C 180,E1 -7697.462,E2 -7697.462} C_VEL
LIN {X 0,Y 467.761,Z 459.412,A -85,B 0,C 180,E1 -7700.02,E2 -7700.02} C_VEL
LIN {X 0,Y 467.837,Z 460.213,A -85,B 0,C 180,E1 -7703.066,E2 -7703.066} C_VEL
LIN {X 0,Y 467.816,Z 461.445,A -85,B 0,C 180,E1 -7705.717,E2 -7705.717} C_VEL
LIN {X 0,Y 467.647,Z 462.959,A -85,B 0,C 180,E1 -7708.265,E2 -7708.265} C_VEL
LIN {X 0,Y 467.463,Z 465.049,A -85,B 0,C 180,E1 -7711.243,E2 -7711.243} C_VEL
LIN {X 0,Y 467.288,Z 467.552,A -85,B 0,C 180,E1 -7714.476,E2 -7714.476} C_VEL
LIN {X 0,Y 467.168,Z 469.646,A -85,B 0,C 180,E1 -7716.975,E2 -7716.975} C_VEL
LIN {X 0,Y 467.058,Z 472.089,A -85,B 0,C 180,E1 -7719.752,E2 -7719.752} C_VEL
LIN {X 0,Y 466.99,Z 474.598,A -85,B 0,C 180,E1 -7722.483,E2 -7722.483} C_VEL
LIN {X 0,Y 467.017,Z 476.743,A -85,B 0,C 180,E1 -7724.739,E2 -7724.739} C_VEL
LIN {X 0,Y 469.978,Z 489.42,A -85,B 0,C 180,E1 -7725.273,E2 -7725.273} C_VEL
LIN {X 0,Y 470.134,Z 495.785,A -85,B 0,C 180,E1 -7725.555,E2 -7725.555} C_VEL
LIN {X 0,Y 469.76,Z 507.117,A -85,B 0,C 180,E1 -7726.151,E2 -7726.151} C_VEL
LIN {X 0,Y 469.327,Z 518.824,A -85,B 0,C 180,E1 -7726.95,E2 -7726.95} C_VEL
LIN {X 0,Y 468.815,Z 529.714,A -85,B 0,C 180,E1 -7727.885,E2 -7727.885} C_VEL
LIN {X 0,Y 468.296,Z 539.912,A -85,B 0,C 180,E1 -7728.969,E2 -7728.969} C_VEL
LIN {X 0,Y 467.847,Z 549.675,A -85,B 0,C 180,E1 -7730.271,E2 -7730.271} C_VEL
LIN {X 0,Y 467.45,Z 557.526,A -85,B 0,C 180,E1 -7731.571,E2 -7731.571} C_VEL
LIN {X 0,Y 467.22,Z 562.822,A -85,B 0,C 180,E1 -7732.654,E2 -7732.654} C_VEL
LIN {X 0,Y 467.057,Z 567.987,A -85,B 0,C 180,E1 -7733.954,E2 -7733.954} C_VEL
LIN {X 0,Y 466.887,Z 571.984,A -85,B 0,C 180,E1 -7735.251,E2 -7735.251} C_VEL
LIN {X 0,Y 466.793,Z 574.921,A -85,B 0,C 180,E1 -7736.548,E2 -7736.548} C_VEL
LIN {X 0,Y 466.809,Z 576.332,A -85,B 0,C 180,E1 -7737.411,E2 -7737.411} C_VEL
LIN {X 0,Y 466.62,Z 577.923,A -85,B 0,C 180,E1 -7739.137,E2 -7739.137} C_VEL
LIN {X 0,Y 466.6,Z 578.133,A -85,B 0,C 180,E1 -7740,E2 -7740} C_VEL
LIN {X 0,Y 466.62,Z 577.913,A -85,B 0,C 180,E1 -7740.863,E2 -7740.863} C_VEL
LIN {X 0,Y 466.79,Z 576.267,A -85,B 0,C 180,E1 -7742.589,E2 -7742.589} C_VEL
LIN {X 0,Y 466.786,Z 574.855,A -85,B 0,C 180,E1 -7743.453,E2 -7743.453} C_VEL
LIN {X 0,Y 466.86,Z 571.894,A -85,B 0,C 180,E1 -7744.75,E2 -7744.75} C_VEL
LIN {X 0,Y 467.045,Z 567.886,A -85,B 0,C 180,E1 -7746.047,E2 -7746.047} C_VEL
LIN {X 0,Y 467.173,Z 562.727,A -85,B 0,C 180,E1 -7747.347,E2 -7747.347} C_VEL
LIN {X 0,Y 467.43,Z 556.22,A -85,B 0,C 180,E1 -7748.648,E2 -7748.648} C_VEL
LIN {X 0,Y 467.788,Z 548.123,A -85,B 0,C 180,E1 -7749.949,E2 -7749.949} C_VEL
LIN {X 0,Y 468.17,Z 539.866,A -85,B 0,C 180,E1 -7751.035,E2 -7751.035} C_VEL
LIN {X 0,Y 468.738,Z 529.781,A -85,B 0,C 180,E1 -7752.117,E2 -7752.117} C_VEL
LIN {X 0,Y 469.142,Z 518.266,A -85,B 0,C 180,E1 -7753.107,E2 -7753.107} C_VEL
LIN {X 0,Y 469.554,Z 507.32,A -85,B 0,C 180,E1 -7753.856,E2 -7753.856} C_VEL
LIN {X 0,Y 469.986,Z 495.028,A -85,B 0,C 180,E1 -7754.506,E2 -7754.506} C_VEL
LIN {X 0,Y 469.852,Z 489.361,A -85,B 0,C 180,E1 -7754.754,E2 -7754.754} C_VEL
LIN {X 0,Y 467.679,Z 478.771,A -85,B 0,C 180,E1 -7755.187,E2 -7755.187} C_VEL
LIN {X 0,Y 466.852,Z 474.833,A -85,B 0,C 180,E1 -7755.323,E2 -7755.323} C_VEL
LIN {X 0,Y 466.829,Z 471.352,A -85,B 0,C 180,E1 -7758.477,E2 -7758.477} C_VEL
LIN {X 0,Y 466.807,Z 468.406,A -85,B 0,C 180,E1 -7761.182,E2 -7761.182} C_VEL
LIN {X 0,Y 466.862,Z 465.394,A -85,B 0,C 180,E1 -7763.982,E2 -7763.982} C_VEL
LIN {X 0,Y 466.948,Z 462.367,A -85,B 0,C 180,E1 -7766.842,E2 -7766.842} C_VEL
LIN {X 0,Y 466.958,Z 459.298,A -85,B 0,C 180,E1 -7769.78,E2 -7769.78} C_VEL
LIN {X 0,Y 467.012,Z 458.318,A -85,B 0,C 180,E1 -7770.931,E2 -7770.931} C_VEL
LIN {X 0,Y 467.395,Z 458.269,A -85,B 0,C 180,E1 -7774.207,E2 -7774.207} C_VEL
LIN {X 0,Y 467.543,Z 458.246,A -85,B 0,C 180,E1 -7777.185,E2 -7777.185} C_VEL
LIN {X 0,Y 467.58,Z 458.244,A -85,B 0,C 180,E1 -7780.265,E2 -7780.265} C_VEL
LIN {X 0,Y 467.591,Z 458.239,A -85,B 0,C 180,E1 -7782.567,E2 -7782.567} C_VEL
LIN {X 0,Y 467.575,Z 458.242,A -85,B 0,C 180,E1 -7785.053,E2 -7785.053} C_VEL
LIN {X 0,Y 467.593,Z 458.241,A -85,B 0,C 180,E1 -7787.44,E2 -7787.44} C_VEL
LIN {X 0,Y 467.587,Z 458.241,A -85,B 0,C 180,E1 -7790.856,E2 -7790.856} C_VEL
LIN {X 0,Y 467.565,Z 458.246,A -85,B 0,C 180,E1 -7794.261,E2 -7794.261} C_VEL
LIN {X 0,Y 467.587,Z 458.241,A -85,B 0,C 180,E1 -7797.321,E2 -7797.321} C_VEL
LIN {X 0,Y 467.575,Z 458.244,A -85,B 0,C 180,E1 -7800.667,E2 -7800.667} C_VEL
LIN {X 0,Y 467.618,Z 458.236,A -85,B 0,C 180,E1 -7803.2,E2 -7803.2} C_VEL
LIN {X 0,Y 467.596,Z 458.239,A -85,B 0,C 180,E1 -7806.469,E2 -7806.469} C_VEL
LIN {X 0,Y 467.628,Z 458.238,A -85,B 0,C 180,E1 -7809.777,E2 -7809.777} C_VEL
LIN {X 0,Y 467.622,Z 458.237,A -85,B 0,C 180,E1 -7811.424,E2 -7811.424} C_VEL
LIN {X 0,Y 466.979,Z 458.32,A -85,B 0,C 180,E1 -7812.143,E2 -7812.143} C_VEL
LIN {X 0,Y 464.131,Z 458.675,A -85,B 0,C 180,E1 -7813.311,E2 -7813.311} C_VEL
LIN {X 0,Y 461.701,Z 458.976,A -85,B 0,C 180,E1 -7814.253,E2 -7814.253} C_VEL
LIN {X 0,Y 460.647,Z 459.105,A -85,B 0,C 180,E1 -7814.981,E2 -7814.981} C_VEL
LIN {X 0,Y 460.556,Z 459.115,A -85,B 0,C 180,E1 -7815.227,E2 -7815.227} C_VEL
LIN {X 0,Y 460.616,Z 459.107,A -85,B 0,C 180,E1 -7818.559,E2 -7818.559} C_VEL
LIN {X 0,Y 460.701,Z 459.098,A -85,B 0,C 180,E1 -7822.109,E2 -7822.109} C_VEL
LIN {X 0,Y 460.702,Z 459.099,A -85,B 0,C 180,E1 -7824.748,E2 -7824.748} C_VEL
LIN {X 0,Y 460.806,Z 459.085,A -85,B 0,C 180,E1 -7827.378,E2 -7827.378} C_VEL
LIN {X 0,Y 460.859,Z 459.081,A -85,B 0,C 180,E1 -7830,E2 -7830} C_VEL
LIN {X 0,Y 460.805,Z 459.083,A -85,B 0,C 180,E1 -7832.622,E2 -7832.622} C_VEL
LIN {X 0,Y 460.691,Z 459.099,A -85,B 0,C 180,E1 -7836.13,E2 -7836.13} C_VEL
LIN {X 0,Y 460.625,Z 459.108,A -85,B 0,C 180,E1 -7838.776,E2 -7838.776} C_VEL
LIN {X 0,Y 460.619,Z 459.108,A -85,B 0,C 180,E1 -7842.445,E2 -7842.445} C_VEL
LIN {X 0,Y 460.606,Z 459.111,A -85,B 0,C 180,E1 -7845.997,E2 -7845.997} C_VEL
LIN {X 0,Y 460.576,Z 459.114,A -85,B 0,C 180,E1 -7848.902,E2 -7848.902} C_VEL
LIN {X 0,Y 460.521,Z 459.12,A -85,B 0,C 180,E1 -7851.485,E2 -7851.485} C_VEL
LIN {X 0,Y 460.536,Z 459.119,A -85,B 0,C 180,E1 -7854.333,E2 -7854.333} C_VEL
LIN {X 0,Y 460.576,Z 459.112,A -85,B 0,C 180,E1 -7857.244,E2 -7857.244} C_VEL
LIN {X 0,Y 460.516,Z 459.12,A -85,B 0,C 180,E1 -7860.24,E2 -7860.24} C_VEL
LIN {X 0,Y 460.534,Z 459.119,A -85,B 0,C 180,E1 -7863.325,E2 -7863.325} C_VEL
LIN {X 0,Y 460.483,Z 459.125,A -85,B 0,C 180,E1 -7866.529,E2 -7866.529} C_VEL
LIN {X 0,Y 460.562,Z 459.117,A -85,B 0,C 180,E1 -7869.859,E2 -7869.859} C_VEL
LIN {X 0,Y 460.518,Z 459.121,A -85,B 0,C 180,E1 -7872.9,E2 -7872.9} C_VEL
LIN {X 0,Y 460.524,Z 459.12,A -85,B 0,C 180,E1 -7875.829,E2 -7875.829} C_VEL
LIN {X 0,Y 460.538,Z 459.117,A -85,B 0,C 180,E1 -7878.989,E2 -7878.989} C_VEL
LIN {X 0,Y 460.53,Z 459.118,A -85,B 0,C 180,E1 -7881.267,E2 -7881.267} C_VEL
LIN {X 0,Y 460.455,Z 459.128,A -85,B 0,C 180,E1 -7884.549,E2 -7884.549} C_VEL
LIN {X 0,Y 460.274,Z 459.154,A -85,B 0,C 180,E1 -7887.12,E2 -7887.12} C_VEL
LIN {X 0,Y 459.906,Z 459.201,A -85,B 0,C 180,E1 -7889.716,E2 -7889.716} C_VEL
LIN {X 0,Y 459.782,Z 459.217,A -85,B 0,C 180,E1 -7890.716,E2 -7890.716} C_VEL
LIN {X 0,Y 459.811,Z 462.549,A -85,B 0,C 180,E1 -7893.688,E2 -7893.688} C_VEL
LIN {X 0,Y 459.734,Z 465.846,A -85,B 0,C 180,E1 -7896.58,E2 -7896.58} C_VEL
LIN {X 0,Y 459.721,Z 469.074,A -85,B 0,C 180,E1 -7899.414,E2 -7899.414} C_VEL
LIN {X 0,Y 459.666,Z 472.271,A -85,B 0,C 180,E1 -7902.194,E2 -7902.194} C_VEL
LIN {X 0,Y 459.678,Z 474.977,A -85,B 0,C 180,E1 -7904.556,E2 -7904.556} C_VEL
LIN {X 0,Y 462.641,Z 488.547,A -85,B 0,C 180,E1 -7905.09,E2 -7905.09} C_VEL
LIN {X 0,Y 463.178,Z 492.588,A -85,B 0,C 180,E1 -7905.276,E2 -7905.276} C_VEL
LIN {X 0,Y 462.696,Z 505.539,A -85,B 0,C 180,E1 -7905.934,E2 -7905.934} C_VEL
LIN {X 0,Y 462.3,Z 517.102,A -85,B 0,C 180,E1 -7906.708,E2 -7906.708} C_VEL
LIN {X 0,Y 461.866,Z 527.608,A -85,B 0,C 180,E1 -7907.588,E2 -7907.588} C_VEL
LIN {X 0,Y 461.312,Z 537.204,A -85,B 0,C 180,E1 -7908.577,E2 -7908.577} C_VEL
LIN {X 0,Y 460.903,Z 545.987,A -85,B 0,C 180,E1 -7909.678,E2 -7909.678} C_VEL
LIN {X 0,Y 460.51,Z 554.595,A -85,B 0,C 180,E1 -7911,E2 -7911} C_VEL
LIN {X 0,Y 460.154,Z 561.458,A -85,B 0,C 180,E1 -7912.32,E2 -7912.32} C_VEL
LIN {X 0,Y 459.997,Z 567.749,A -85,B 0,C 180,E1 -7913.86,E2 -7913.86} C_VEL
LIN {X 0,Y 459.764,Z 571.87,A -85,B 0,C 180,E1 -7915.177,E2 -7915.177} C_VEL
LIN {X 0,Y 459.726,Z 574.921,A -85,B 0,C 180,E1 -7916.494,E2 -7916.494} C_VEL
LIN {X 0,Y 459.692,Z 576.422,A -85,B 0,C 180,E1 -7917.371,E2 -7917.371} C_VEL
LIN {X 0,Y 459.636,Z 577.475,A -85,B 0,C 180,E1 -7918.247,E2 -7918.247} C_VEL
LIN {X 0,Y 459.532,Z 578.426,A -85,B 0,C 180,E1 -7920,E2 -7920} C_VEL
LIN {X 0,Y 459.554,Z 578.266,A -85,B 0,C 180,E1 -7920.876,E2 -7920.876} C_VEL
LIN {X 0,Y 459.736,Z 576.747,A -85,B 0,C 180,E1 -7922.628,E2 -7922.628} C_VEL
LIN {X 0,Y 459.733,Z 575.385,A -85,B 0,C 180,E1 -7923.506,E2 -7923.506} C_VEL
LIN {X 0,Y 459.807,Z 572.508,A -85,B 0,C 180,E1 -7924.822,E2 -7924.822} C_VEL
LIN {X 0,Y 460.003,Z 568.57,A -85,B 0,C 180,E1 -7926.139,E2 -7926.139} C_VEL
LIN {X 0,Y 460.17,Z 563.46,A -85,B 0,C 180,E1 -7927.459,E2 -7927.459} C_VEL
LIN {X 0,Y 460.574,Z 555.843,A -85,B 0,C 180,E1 -7928.998,E2 -7928.998} C_VEL
LIN {X 0,Y 460.944,Z 547.541,A -85,B 0,C 180,E1 -7930.32,E2 -7930.32} C_VEL
LIN {X 0,Y 461.329,Z 539.037,A -85,B 0,C 180,E1 -7931.423,E2 -7931.423} C_VEL
LIN {X 0,Y 461.955,Z 528.617,A -85,B 0,C 180,E1 -7932.521,E2 -7932.521} C_VEL
LIN {X 0,Y 462.418,Z 516.855,A -85,B 0,C 180,E1 -7933.506,E2 -7933.506} C_VEL
LIN {X 0,Y 462.958,Z 505.071,A -85,B 0,C 180,E1 -7934.281,E2 -7934.281} C_VEL
LIN {X 0,Y 463.32,Z 491.675,A -85,B 0,C 180,E1 -7934.944,E2 -7934.944} C_VEL
LIN {X 0,Y 460.832,Z 480.477,A -85,B 0,C 180,E1 -7935.454,E2 -7935.454} C_VEL
LIN {X 0,Y 459.848,Z 476.692,A -85,B 0,C 180,E1 -7935.605,E2 -7935.605} C_VEL
LIN {X 0,Y 459.87,Z 473.117,A -85,B 0,C 180,E1 -7938.719,E2 -7938.719} C_VEL
LIN {X 0,Y 459.831,Z 469.863,A -85,B 0,C 180,E1 -7941.519,E2 -7941.519} C_VEL
LIN {X 0,Y 459.875,Z 466.552,A -85,B 0,C 180,E1 -7944.37,E2 -7944.37} C_VEL
LIN {X 0,Y 459.911,Z 462.868,A -85,B 0,C 180,E1 -7947.286,E2 -7947.286} C_VEL
LIN {X 0,Y 459.85,Z 460.039,A -85,B 0,C 180,E1 -7949.407,E2 -7949.407} C_VEL
LIN {X 0,Y 459.894,Z 459.203,A -85,B 0,C 180,E1 -7950.285,E2 -7950.285} C_VEL
LIN {X 0,Y 460.317,Z 459.149,A -85,B 0,C 180,E1 -7953.342,E2 -7953.342} C_VEL
LIN {X 0,Y 460.482,Z 459.128,A -85,B 0,C 180,E1 -7956.011,E2 -7956.011} C_VEL
LIN {X 0,Y 460.546,Z 459.118,A -85,B 0,C 180,E1 -7958.898,E2 -7958.898} C_VEL
LIN {X 0,Y 460.526,Z 459.123,A -85,B 0,C 180,E1 -7962.181,E2 -7962.181} C_VEL
LIN {X 0,Y 460.519,Z 459.122,A -85,B 0,C 180,E1 -7965.411,E2 -7965.411} C_VEL
LIN {X 0,Y 460.534,Z 459.121,A -85,B 0,C 180,E1 -7968.397,E2 -7968.397} C_VEL
LIN {X 0,Y 460.567,Z 459.198,A -85,B 0,C 180,E1 -7969.188,E2 -7969.188} C_VEL
LIN {X 0,Y 461.789,Z 466.101,A -85,B 0,C 180,E1 -7972.316,E2 -7972.316} C_VEL
LIN {X 0,Y 462.378,Z 470.483,A -85,B 0,C 180,E1 -7974.21,E2 -7974.21} C_VEL
LIN {X 0,Y 462.015,Z 476.849,A -85,B 0,C 180,E1 -7976.796,E2 -7976.796} C_VEL
LIN {X 0,Y 461.55,Z 484.585,A -85,B 0,C 180,E1 -7979.835,E2 -7979.835} C_VEL
LIN {X 0,Y 461.107,Z 492.345,A -85,B 0,C 180,E1 -7982.79,E2 -7982.79} C_VEL
LIN {X 0,Y 460.767,Z 500.115,A -85,B 0,C 180,E1 -7985.68,E2 -7985.68} C_VEL
LIN {X 0,Y 460.392,Z 509.329,A -85,B 0,C 180,E1 -7989.02,E2 -7989.02} C_VEL
LIN {X 0,Y 460.129,Z 518.307,A -85,B 0,C 180,E1 -7992.213,E2 -7992.213} C_VEL
LIN {X 0,Y 460.031,Z 524.593,A -85,B 0,C 180,E1 -7994.405,E2 -7994.405} C_VEL
LIN {X 0,Y 461.907,Z 538.256,A -85,B 0,C 180,E1 -7994.852,E2 -7994.852} C_VEL
LIN {X 0,Y 462.908,Z 546.393,A -85,B 0,C 180,E1 -7995.211,E2 -7995.211} C_VEL
LIN {X 0,Y 462.425,Z 558.296,A -85,B 0,C 180,E1 -7995.814,E2 -7995.814} C_VEL
LIN {X 0,Y 461.945,Z 569.983,A -85,B 0,C 180,E1 -7996.584,E2 -7996.584} C_VEL
LIN {X 0,Y 461.402,Z 581.289,A -85,B 0,C 180,E1 -7997.534,E2 -7997.534} C_VEL
LIN {X 0,Y 460.93,Z 591.246,A -85,B 0,C 180,E1 -7998.567,E2 -7998.567} C_VEL
LIN {X 0,Y 460.462,Z 599.964,A -85,B 0,C 180,E1 -7999.669,E2 -7999.669} C_VEL
LIN {X 0,Y 460.108,Z 608.448,A -85,B 0,C 180,E1 -8000.992,E2 -8000.992} C_VEL
LIN {X 0,Y 459.868,Z 615.275,A -85,B 0,C 180,E1 -8002.315,E2 -8002.315} C_VEL
LIN {X 0,Y 459.677,Z 621.541,A -85,B 0,C 180,E1 -8003.856,E2 -8003.856} C_VEL
LIN {X 0,Y 459.631,Z 625.602,A -85,B 0,C 180,E1 -8005.176,E2 -8005.176} C_VEL
LIN {X 0,Y 459.627,Z 628.591,A -85,B 0,C 180,E1 -8006.493,E2 -8006.493} C_VEL
LIN {X 0,Y 459.621,Z 630.019,A -85,B 0,C 180,E1 -8007.371,E2 -8007.371} C_VEL
LIN {X 0,Y 459.629,Z 631.022,A -85,B 0,C 180,E1 -8008.248,E2 -8008.248} C_VEL
LIN {X 0,Y 459.553,Z 631.62,A -85,B 0,C 180,E1 -8009.124,E2 -8009.124} C_VEL
LIN {X 0,Y 459.529,Z 631.819,A -85,B 0,C 180,E1 -8010,E2 -8010} C_VEL
LIN {X 0,Y 459.553,Z 631.571,A -85,B 0,C 180,E1 -8010.876,E2 -8010.876} C_VEL
LIN {X 0,Y 459.631,Z 630.919,A -85,B 0,C 180,E1 -8011.752,E2 -8011.752} C_VEL
LIN {X 0,Y 459.63,Z 629.858,A -85,B 0,C 180,E1 -8012.629,E2 -8012.629} C_VEL
LIN {X 0,Y 459.643,Z 628.379,A -85,B 0,C 180,E1 -8013.506,E2 -8013.506} C_VEL
LIN {X 0,Y 459.631,Z 625.29,A -85,B 0,C 180,E1 -8014.824,E2 -8014.824} C_VEL
LIN {X 0,Y 459.714,Z 620.038,A -85,B 0,C 180,E1 -8016.431,E2 -8016.431} C_VEL
LIN {X 0,Y 459.894,Z 613.685,A -85,B 0,C 180,E1 -8017.905,E2 -8017.905} C_VEL
LIN {X 0,Y 460.181,Z 606.486,A -85,B 0,C 180,E1 -8019.228,E2 -8019.228} C_VEL
LIN {X 0,Y 460.507,Z 597.483,A -85,B 0,C 180,E1 -8020.553,E2 -8020.553} C_VEL
LIN {X 0,Y 461.071,Z 587.328,A -85,B 0,C 180,E1 -8021.764,E2 -8021.764} C_VEL
LIN {X 0,Y 461.488,Z 576.918,A -85,B 0,C 180,E1 -8022.767,E2 -8022.767} C_VEL
LIN {X 0,Y 462.002,Z 565.747,A -85,B 0,C 180,E1 -8023.638,E2 -8023.638} C_VEL
LIN {X 0,Y 462.583,Z 553.272,A -85,B 0,C 180,E1 -8024.406,E2 -8024.406} C_VEL
LIN {X 0,Y 462.794,Z 545.371,A -85,B 0,C 180,E1 -8024.792,E2 -8024.792} C_VEL
LIN {X 0,Y 461.169,Z 531.719,A -85,B 0,C 180,E1 -8025.377,E2 -8025.377} C_VEL
LIN {X 0,Y 459.944,Z 522.74,A -85,B 0,C 180,E1 -8025.664,E2 -8025.664} C_VEL
LIN {X 0,Y 460.125,Z 512.627,A -85,B 0,C 180,E1 -8029.125,E2 -8029.125} C_VEL
LIN {X 0,Y 460.346,Z 504.579,A -85,B 0,C 180,E1 -8031.965,E2 -8031.965} C_VEL
LIN {X 0,Y 460.678,Z 495.558,A -85,B 0,C 180,E1 -8035.288,E2 -8035.288} C_VEL
LIN {X 0,Y 461.042,Z 488.123,A -85,B 0,C 180,E1 -8038.2,E2 -8038.2} C_VEL
LIN {X 0,Y 461.591,Z 480.372,A -85,B 0,C 180,E1 -8041.501,E2 -8041.501} C_VEL
LIN {X 0,Y 462.143,Z 474.635,A -85,B 0,C 180,E1 -8044.241,E2 -8044.241} C_VEL
LIN {X 0,Y 462.399,Z 470.78,A -85,B 0,C 180,E1 -8046.353,E2 -8046.353} C_VEL
LIN {X 0,Y 462.013,Z 467.441,A -85,B 0,C 180,E1 -8048.586,E2 -8048.586} C_VEL
LIN {X 0,Y 461.528,Z 464.7,A -85,B 0,C 180,E1 -8050.904,E2 -8050.904} C_VEL
LIN {X 0,Y 461.141,Z 462.652,A -85,B 0,C 180,E1 -8053.3,E2 -8053.3} C_VEL
LIN {X 0,Y 460.922,Z 461.349,A -85,B 0,C 180,E1 -8055.778,E2 -8055.778} C_VEL
LIN {X 0,Y 460.825,Z 460.803,A -85,B 0,C 180,E1 -8058.357,E2 -8058.357} C_VEL
LIN {X 0,Y 460.804,Z 461.043,A -85,B 0,C 180,E1 -8061.295,E2 -8061.295} C_VEL
LIN {X 0,Y 460.869,Z 461.851,A -85,B 0,C 180,E1 -8063.923,E2 -8063.923} C_VEL
LIN {X 0,Y 460.746,Z 463.376,A -85,B 0,C 180,E1 -8067.029,E2 -8067.029} C_VEL
LIN {X 0,Y 460.511,Z 465.551,A -85,B 0,C 180,E1 -8070.447,E2 -8070.447} C_VEL
LIN {X 0,Y 460.287,Z 467.945,A -85,B 0,C 180,E1 -8073.718,E2 -8073.718} C_VEL
LIN {X 0,Y 460.181,Z 470.267,A -85,B 0,C 180,E1 -8076.604,E2 -8076.604} C_VEL
LIN {X 0,Y 460.019,Z 472.686,A -85,B 0,C 180,E1 -8079.428,E2 -8079.428} C_VEL
LIN {X 0,Y 459.945,Z 475.185,A -85,B 0,C 180,E1 -8082.206,E2 -8082.206} C_VEL
LIN {X 0,Y 459.946,Z 477.301,A -85,B 0,C 180,E1 -8084.471,E2 -8084.471} C_VEL
LIN {X 0,Y 463.097,Z 490.22,A -85,B 0,C 180,E1 -8085.049,E2 -8085.049} C_VEL
LIN {X 0,Y 463.309,Z 495.315,A -85,B 0,C 180,E1 -8085.281,E2 -8085.281} C_VEL
LIN {X 0,Y 462.916,Z 507.758,A -85,B 0,C 180,E1 -8085.942,E2 -8085.942} C_VEL
LIN {X 0,Y 462.45,Z 518.391,A -85,B 0,C 180,E1 -8086.67,E2 -8086.67} C_VEL
LIN {X 0,Y 461.901,Z 530.268,A -85,B 0,C 180,E1 -8087.701,E2 -8087.701} C_VEL
LIN {X 0,Y 461.344,Z 540.431,A -85,B 0,C 180,E1 -8088.8,E2 -8088.8} C_VEL
LIN {X 0,Y 460.868,Z 550.145,A -85,B 0,C 180,E1 -8090.122,E2 -8090.122} C_VEL
LIN {X 0,Y 460.438,Z 557.967,A -85,B 0,C 180,E1 -8091.442,E2 -8091.442} C_VEL
LIN {X 0,Y 460.185,Z 563.247,A -85,B 0,C 180,E1 -8092.541,E2 -8092.541} C_VEL
LIN {X 0,Y 460.016,Z 568.417,A -85,B 0,C 180,E1 -8093.861,E2 -8093.861} C_VEL
LIN {X 0,Y 459.83,Z 572.417,A -85,B 0,C 180,E1 -8095.178,E2 -8095.178} C_VEL
LIN {X 0,Y 459.733,Z 575.353,A -85,B 0,C 180,E1 -8096.494,E2 -8096.494} C_VEL
LIN {X 0,Y 459.736,Z 576.763,A -85,B 0,C 180,E1 -8097.372,E2 -8097.372} C_VEL
LIN {X 0,Y 459.554,Z 578.344,A -85,B 0,C 180,E1 -8099.124,E2 -8099.124} C_VEL
LIN {X 0,Y 459.531,Z 578.549,A -85,B 0,C 180,E1 -8100,E2 -8100} C_VEL
LIN {X 0,Y 459.554,Z 578.319,A -85,B 0,C 180,E1 -8100.876,E2 -8100.876} C_VEL
LIN {X 0,Y 459.637,Z 577.682,A -85,B 0,C 180,E1 -8101.753,E2 -8101.753} C_VEL
LIN {X 0,Y 459.705,Z 576.654,A -85,B 0,C 180,E1 -8102.629,E2 -8102.629} C_VEL
LIN {X 0,Y 459.725,Z 575.229,A -85,B 0,C 180,E1 -8103.506,E2 -8103.506} C_VEL
LIN {X 0,Y 459.789,Z 572.247,A -85,B 0,C 180,E1 -8104.823,E2 -8104.823} C_VEL
LIN {X 0,Y 460.004,Z 568.213,A -85,B 0,C 180,E1 -8106.14,E2 -8106.14} C_VEL
LIN {X 0,Y 460.157,Z 562.011,A -85,B 0,C 180,E1 -8107.68,E2 -8107.68} C_VEL
LIN {X 0,Y 460.504,Z 555.24,A -85,B 0,C 180,E1 -8109,E2 -8109} C_VEL
LIN {X 0,Y 460.885,Z 546.841,A -85,B 0,C 180,E1 -8110.322,E2 -8110.322} C_VEL
LIN {X 0,Y 461.275,Z 538.195,A -85,B 0,C 180,E1 -8111.424,E2 -8111.424} C_VEL
LIN {X 0,Y 461.901,Z 527.691,A -85,B 0,C 180,E1 -8112.512,E2 -8112.512} C_VEL
LIN {X 0,Y 462.281,Z 517.091,A -85,B 0,C 180,E1 -8113.406,E2 -8113.406} C_VEL
LIN {X 0,Y 462.748,Z 505.515,A -85,B 0,C 180,E1 -8114.176,E2 -8114.176} C_VEL
LIN {X 0,Y 463.204,Z 492.473,A -85,B 0,C 180,E1 -8114.835,E2 -8114.835} C_VEL
LIN {X 0,Y 461.988,Z 485.133,A -85,B 0,C 180,E1 -8115.169,E2 -8115.169} C_VEL
LIN {X 0,Y 459.762,Z 475.138,A -85,B 0,C 180,E1 -8115.574,E2 -8115.574} C_VEL
LIN {X 0,Y 459.736,Z 471.673,A -85,B 0,C 180,E1 -8118.725,E2 -8118.725} C_VEL
LIN {X 0,Y 459.743,Z 468.648,A -85,B 0,C 180,E1 -8121.524,E2 -8121.524} C_VEL
LIN {X 0,Y 459.804,Z 465.601,A -85,B 0,C 180,E1 -8124.374,E2 -8124.374} C_VEL
LIN {X 0,Y 459.917,Z 462.535,A -85,B 0,C 180,E1 -8127.286,E2 -8127.286} C_VEL
LIN {X 0,Y 459.903,Z 459.432,A -85,B 0,C 180,E1 -8130.285,E2 -8130.285} C_VEL
LIN {X 0,Y 460.173,Z 459.168,A -85,B 0,C 180,E1 -8132.861,E2 -8132.861} C_VEL
LIN {X 0,Y 460.442,Z 459.131,A -85,B 0,C 180,E1 -8135.452,E2 -8135.452} C_VEL
LIN {X 0,Y 460.522,Z 459.122,A -85,B 0,C 180,E1 -8138.734,E2 -8138.734} C_VEL
LIN {X 0,Y 460.539,Z 459.116,A -85,B 0,C 180,E1 -8141.603,E2 -8141.603} C_VEL
LIN {X 0,Y 460.525,Z 459.119,A -85,B 0,C 180,E1 -8144.588,E2 -8144.588} C_VEL
LIN {X 0,Y 460.527,Z 459.12,A -85,B 0,C 180,E1 -8147.819,E2 -8147.819} C_VEL
LIN {X 0,Y 460.549,Z 459.116,A -85,B 0,C 180,E1 -8151.102,E2 -8151.102} C_VEL
LIN {X 0,Y 460.515,Z 459.121,A -85,B 0,C 180,E1 -8154.555,E2 -8154.555} C_VEL
LIN {X 0,Y 460.536,Z 459.121,A -85,B 0,C 180,E1 -8157.716,E2 -8157.716} C_VEL
LIN {X 0,Y 460.545,Z 459.119,A -85,B 0,C 180,E1 -8160.769,E2 -8160.769} C_VEL
LIN {X 0,Y 460.561,Z 459.114,A -85,B 0,C 180,E1 -8163.734,E2 -8163.734} C_VEL
LIN {X 0,Y 460.55,Z 459.116,A -85,B 0,C 180,E1 -8166.624,E2 -8166.624} C_VEL
LIN {X 0,Y 460.557,Z 459.116,A -85,B 0,C 180,E1 -8169.453,E2 -8169.453} C_VEL
LIN {X 0,Y 460.555,Z 459.116,A -85,B 0,C 180,E1 -8172.23,E2 -8172.23} C_VEL
LIN {X 0,Y 460.571,Z 459.114,A -85,B 0,C 180,E1 -8174.965,E2 -8174.965} C_VEL
LIN {X 0,Y 460.556,Z 459.115,A -85,B 0,C 180,E1 -8175.227,E2 -8175.227} C_VEL
LIN {X 0,Y 459.878,Z 459.202,A -85,B 0,C 180,E1 -8175.957,E2 -8175.957} C_VEL
LIN {X 0,Y 457.031,Z 459.553,A -85,B 0,C 180,E1 -8177.143,E2 -8177.143} C_VEL
LIN {X 0,Y 454.634,Z 459.857,A -85,B 0,C 180,E1 -8178.1,E2 -8178.1} C_VEL
LIN {X 0,Y 453.612,Z 459.979,A -85,B 0,C 180,E1 -8178.839,E2 -8178.839} C_VEL
LIN {X 0,Y 453.532,Z 459.988,A -85,B 0,C 180,E1 -8179.089,E2 -8179.089} C_VEL
LIN {X 0,Y 453.699,Z 459.97,A -85,B 0,C 180,E1 -8182.48,E2 -8182.48} C_VEL
LIN {X 0,Y 453.675,Z 459.975,A -85,B 0,C 180,E1 -8184.667,E2 -8184.667} C_VEL
LIN {X 0,Y 453.75,Z 459.964,A -85,B 0,C 180,E1 -8187.337,E2 -8187.337} C_VEL
LIN {X 0,Y 453.829,Z 459.956,A -85,B 0,C 180,E1 -8190,E2 -8190} C_VEL
LIN {X 0,Y 453.749,Z 459.962,A -85,B 0,C 180,E1 -8192.663,E2 -8192.663} C_VEL
LIN {X 0,Y 453.657,Z 459.975,A -85,B 0,C 180,E1 -8196.226,E2 -8196.226} C_VEL
LIN {X 0,Y 453.591,Z 459.984,A -85,B 0,C 180,E1 -8198.913,E2 -8198.913} C_VEL
LIN {X 0,Y 453.569,Z 459.985,A -85,B 0,C 180,E1 -8202.529,E2 -8202.529} C_VEL
LIN {X 0,Y 453.55,Z 459.988,A -85,B 0,C 180,E1 -8206.196,E2 -8206.196} C_VEL
LIN {X 0,Y 453.526,Z 459.992,A -85,B 0,C 180,E1 -8209.041,E2 -8209.041} C_VEL
LIN {X 0,Y 453.482,Z 459.997,A -85,B 0,C 180,E1 -8211.836,E2 -8211.836} C_VEL
LIN {X 0,Y 453.506,Z 459.993,A -85,B 0,C 180,E1 -8214.735,E2 -8214.735} C_VEL
LIN {X 0,Y 453.537,Z 459.991,A -85,B 0,C 180,E1 -8217.959,E2 -8217.959} C_VEL
LIN {X 0,Y 453.471,Z 460,A -85,B 0,C 180,E1 -8221.525,E2 -8221.525} C_VEL
LIN {X 0,Y 453.494,Z 459.996,A -85,B 0,C 180,E1 -8224.777,E2 -8224.777} C_VEL
LIN {X 0,Y 453.477,Z 459.997,A -85,B 0,C 180,E1 -8228.311,E2 -8228.311} C_VEL
LIN {X 0,Y 453.498,Z 459.993,A -85,B 0,C 180,E1 -8230.609,E2 -8230.609} C_VEL
LIN {X 0,Y 453.461,Z 460.002,A -85,B 0,C 180,E1 -8233.244,E2 -8233.244} C_VEL
LIN {X 0,Y 453.478,Z 459.998,A -85,B 0,C 180,E1 -8235.78,E2 -8235.78} C_VEL
LIN {X 0,Y 453.486,Z 459.998,A -85,B 0,C 180,E1 -8238.209,E2 -8238.209} C_VEL
LIN {X 0,Y 453.498,Z 459.992,A -85,B 0,C 180,E1 -8240.793,E2 -8240.793} C_VEL
LIN {X 0,Y 453.424,Z 460.004,A -85,B 0,C 180,E1 -8243.914,E2 -8243.914} C_VEL
LIN {X 0,Y 453.276,Z 460.024,A -85,B 0,C 180,E1 -8246.853,E2 -8246.853} C_VEL
LIN {X 0,Y 452.779,Z 460.089,A -85,B 0,C 180,E1 -8250.369,E2 -8250.369} C_VEL
LIN {X 0,Y 452.704,Z 460.339,A -85,B 0,C 180,E1 -8251.232,E2 -8251.232} C_VEL
LIN {X 0,Y 452.721,Z 463.763,A -85,B 0,C 180,E1 -8254.235,E2 -8254.235} C_VEL
LIN {X 0,Y 452.625,Z 467.099,A -85,B 0,C 180,E1 -8257.158,E2 -8257.158} C_VEL
LIN {X 0,Y 452.64,Z 470.362,A -85,B 0,C 180,E1 -8260.026,E2 -8260.026} C_VEL
LIN {X 0,Y 452.573,Z 473.578,A -85,B 0,C 180,E1 -8262.839,E2 -8262.839} C_VEL
LIN {X 0,Y 452.601,Z 475.262,A -85,B 0,C 180,E1 -8264.311,E2 -8264.311} C_VEL
LIN {X 0,Y 455.785,Z 489.816,A -85,B 0,C 180,E1 -8264.917,E2 -8264.917} C_VEL
LIN {X 0,Y 456.254,Z 493.794,A -85,B 0,C 180,E1 -8265.105,E2 -8265.105} C_VEL
LIN {X 0,Y 455.806,Z 505.551,A -85,B 0,C 180,E1 -8265.717,E2 -8265.717} C_VEL
LIN {X 0,Y 455.409,Z 516.7,A -85,B 0,C 180,E1 -8266.468,E2 -8266.468} C_VEL
LIN {X 0,Y 454.928,Z 527.778,A -85,B 0,C 180,E1 -8267.4,E2 -8267.4} C_VEL
LIN {X 0,Y 454.358,Z 537.372,A -85,B 0,C 180,E1 -8268.399,E2 -8268.399} C_VEL
LIN {X 0,Y 453.927,Z 546.192,A -85,B 0,C 180,E1 -8269.518,E2 -8269.518} C_VEL
LIN {X 0,Y 453.508,Z 554.838,A -85,B 0,C 180,E1 -8270.86,E2 -8270.86} C_VEL
LIN {X 0,Y 453.135,Z 561.738,A -85,B 0,C 180,E1 -8272.2,E2 -8272.2} C_VEL
LIN {X 0,Y 452.958,Z 568.061,A -85,B 0,C 180,E1 -8273.765,E2 -8273.765} C_VEL
LIN {X 0,Y 452.681,Z 572.208,A -85,B 0,C 180,E1 -8275.101,E2 -8275.101} C_VEL
LIN {X 0,Y 452.667,Z 575.28,A -85,B 0,C 180,E1 -8276.439,E2 -8276.439} C_VEL
LIN {X 0,Y 452.612,Z 576.796,A -85,B 0,C 180,E1 -8277.33,E2 -8277.33} C_VEL
LIN {X 0,Y 452.576,Z 577.859,A -85,B 0,C 180,E1 -8278.22,E2 -8278.22} C_VEL
LIN {X 0,Y 452.466,Z 578.826,A -85,B 0,C 180,E1 -8280,E2 -8280} C_VEL
LIN {X 0,Y 452.49,Z 578.673,A -85,B 0,C 180,E1 -8280.89,E2 -8280.89} C_VEL
LIN {X 0,Y 452.578,Z 578.111,A -85,B 0,C 180,E1 -8281.78,E2 -8281.78} C_VEL
LIN {X 0,Y 452.652,Z 577.164,A -85,B 0,C 180,E1 -8282.67,E2 -8282.67} C_VEL
LIN {X 0,Y 452.675,Z 575.807,A -85,B 0,C 180,E1 -8283.56,E2 -8283.56} C_VEL
LIN {X 0,Y 452.739,Z 572.944,A -85,B 0,C 180,E1 -8284.898,E2 -8284.898} C_VEL
LIN {X 0,Y 453.025,Z 567.957,A -85,B 0,C 180,E1 -8286.538,E2 -8286.538} C_VEL
LIN {X 0,Y 453.231,Z 561.976,A -85,B 0,C 180,E1 -8288.022,E2 -8288.022} C_VEL
LIN {X 0,Y 453.634,Z 555.059,A -85,B 0,C 180,E1 -8289.362,E2 -8289.362} C_VEL
LIN {X 0,Y 454.095,Z 546.461,A -85,B 0,C 180,E1 -8290.703,E2 -8290.703} C_VEL
LIN {X 0,Y 454.58,Z 537.651,A -85,B 0,C 180,E1 -8291.821,E2 -8291.821} C_VEL
LIN {X 0,Y 455.174,Z 526.863,A -85,B 0,C 180,E1 -8292.922,E2 -8292.922} C_VEL
LIN {X 0,Y 455.609,Z 515.892,A -85,B 0,C 180,E1 -8293.833,E2 -8293.833} C_VEL
LIN {X 0,Y 456.195,Z 503.815,A -85,B 0,C 180,E1 -8294.612,E2 -8294.612} C_VEL
LIN {X 0,Y 456.502,Z 492.648,A -85,B 0,C 180,E1 -8295.172,E2 -8295.172} C_VEL
LIN {X 0,Y 453.885,Z 481.31,A -85,B 0,C 180,E1 -8295.717,E2 -8295.717} C_VEL
LIN {X 0,Y 452.799,Z 477.18,A -85,B 0,C 180,E1 -8295.888,E2 -8295.888} C_VEL
LIN {X 0,Y 452.799,Z 473.604,A -85,B 0,C 180,E1 -8299.023,E2 -8299.023} C_VEL
LIN {X 0,Y 452.793,Z 470.313,A -85,B 0,C 180,E1 -8301.871,E2 -8301.871} C_VEL
LIN {X 0,Y 452.84,Z 466.886,A -85,B 0,C 180,E1 -8304.774,E2 -8304.774} C_VEL
LIN {X 0,Y 452.858,Z 464.389,A -85,B 0,C 180,E1 -8306.747,E2 -8306.747} C_VEL
LIN {X 0,Y 452.807,Z 460.529,A -85,B 0,C 180,E1 -8309.78,E2 -8309.78} C_VEL
LIN {X 0,Y 453.024,Z 460.058,A -85,B 0,C 180,E1 -8311.433,E2 -8311.433} C_VEL
LIN {X 0,Y 453.329,Z 460.02,A -85,B 0,C 180,E1 -8313.925,E2 -8313.925} C_VEL
LIN {X 0,Y 453.452,Z 460.003,A -85,B 0,C 180,E1 -8317.19,E2 -8317.19} C_VEL
LIN {X 0,Y 453.519,Z 459.995,A -85,B 0,C 180,E1 -8319.447,E2 -8319.447} C_VEL
LIN {X 0,Y 453.47,Z 460.001,A -85,B 0,C 180,E1 -8322.994,E2 -8322.994} C_VEL
LIN {X 0,Y 453.468,Z 460.002,A -85,B 0,C 180,E1 -8325.779,E2 -8325.779} C_VEL
LIN {X 0,Y 453.524,Z 460.173,A -85,B 0,C 180,E1 -8328.969,E2 -8328.969} C_VEL
LIN {X 0,Y 454.717,Z 466.775,A -85,B 0,C 180,E1 -8332.022,E2 -8332.022} C_VEL
LIN {X 0,Y 455.374,Z 471.472,A -85,B 0,C 180,E1 -8334.093,E2 -8334.093} C_VEL
LIN {X 0,Y 455.063,Z 477.316,A -85,B 0,C 180,E1 -8336.51,E2 -8336.51} C_VEL
LIN {X 0,Y 454.473,Z 486.057,A -85,B 0,C 180,E1 -8339.996,E2 -8339.996} C_VEL
LIN {X 0,Y 454.07,Z 493.374,A -85,B 0,C 180,E1 -8342.832,E2 -8342.832} C_VEL
LIN {X 0,Y 453.624,Z 502.425,A -85,B 0,C 180,E1 -8346.245,E2 -8346.245} C_VEL
LIN {X 0,Y 453.311,Z 510.196,A -85,B 0,C 180,E1 -8349.109,E2 -8349.109} C_VEL
LIN {X 0,Y 453.031,Z 519.274,A -85,B 0,C 180,E1 -8352.392,E2 -8352.392} C_VEL
LIN {X 0,Y 452.937,Z 524.457,A -85,B 0,C 180,E1 -8354.177,E2 -8354.177} C_VEL
LIN {X 0,Y 454.879,Z 538.285,A -85,B 0,C 180,E1 -8354.645,E2 -8354.645} C_VEL
LIN {X 0,Y 455.972,Z 546.897,A -85,B 0,C 180,E1 -8355.038,E2 -8355.038} C_VEL
LIN {X 0,Y 455.436,Z 559.524,A -85,B 0,C 180,E1 -8355.706,E2 -8355.706} C_VEL
LIN {X 0,Y 454.918,Z 570.786,A -85,B 0,C 180,E1 -8356.487,E2 -8356.487} C_VEL
LIN {X 0,Y 454.343,Z 582.318,A -85,B 0,C 180,E1 -8357.493,E2 -8357.493} C_VEL
LIN {X 0,Y 453.927,Z 590.701,A -85,B 0,C 180,E1 -8358.388,E2 -8358.388} C_VEL
LIN {X 0,Y 453.443,Z 599.448,A -85,B 0,C 180,E1 -8359.507,E2 -8359.507} C_VEL
LIN {X 0,Y 453.07,Z 607.969,A -85,B 0,C 180,E1 -8360.851,E2 -8360.851} C_VEL
LIN {X 0,Y 452.782,Z 614.815,A -85,B 0,C 180,E1 -8362.194,E2 -8362.194} C_VEL
LIN {X 0,Y 452.603,Z 621.101,A -85,B 0,C 180,E1 -8363.76,E2 -8363.76} C_VEL
LIN {X 0,Y 452.561,Z 625.176,A -85,B 0,C 180,E1 -8365.1,E2 -8365.1} C_VEL
LIN {X 0,Y 452.527,Z 628.172,A -85,B 0,C 180,E1 -8366.438,E2 -8366.438} C_VEL
LIN {X 0,Y 452.543,Z 629.607,A -85,B 0,C 180,E1 -8367.33,E2 -8367.33} C_VEL
LIN {X 0,Y 452.538,Z 630.61,A -85,B 0,C 180,E1 -8368.22,E2 -8368.22} C_VEL
LIN {X 0,Y 452.489,Z 631.21,A -85,B 0,C 180,E1 -8369.11,E2 -8369.11} C_VEL
LIN {X 0,Y 452.463,Z 631.408,A -85,B 0,C 180,E1 -8370,E2 -8370} C_VEL
LIN {X 0,Y 452.489,Z 631.16,A -85,B 0,C 180,E1 -8370.89,E2 -8370.89} C_VEL
LIN {X 0,Y 452.539,Z 630.501,A -85,B 0,C 180,E1 -8371.78,E2 -8371.78} C_VEL
LIN {X 0,Y 452.552,Z 629.438,A -85,B 0,C 180,E1 -8372.67,E2 -8372.67} C_VEL
LIN {X 0,Y 452.541,Z 627.953,A -85,B 0,C 180,E1 -8373.562,E2 -8373.562} C_VEL
LIN {X 0,Y 452.562,Z 624.857,A -85,B 0,C 180,E1 -8374.9,E2 -8374.9} C_VEL
LIN {X 0,Y 452.628,Z 620.03,A -85,B 0,C 180,E1 -8376.416,E2 -8376.416} C_VEL
LIN {X 0,Y 452.841,Z 613.226,A -85,B 0,C 180,E1 -8378.029,E2 -8378.029} C_VEL
LIN {X 0,Y 453.113,Z 606.023,A -85,B 0,C 180,E1 -8379.373,E2 -8379.373} C_VEL
LIN {X 0,Y 453.495,Z 597.028,A -85,B 0,C 180,E1 -8380.718,E2 -8380.718} C_VEL
LIN {X 0,Y 454.024,Z 586.871,A -85,B 0,C 180,E1 -8381.949,E2 -8381.949} C_VEL
LIN {X 0,Y 454.497,Z 576.499,A -85,B 0,C 180,E1 -8382.967,E2 -8382.967} C_VEL
LIN {X 0,Y 455.163,Z 563.83,A -85,B 0,C 180,E1 -8383.961,E2 -8383.961} C_VEL
LIN {X 0,Y 455.774,Z 550.897,A -85,B 0,C 180,E1 -8384.74,E2 -8384.74} C_VEL
LIN {X 0,Y 455.769,Z 545.228,A -85,B 0,C 180,E1 -8385.026,E2 -8385.026} C_VEL
LIN {X 0,Y 454.237,Z 531.254,A -85,B 0,C 180,E1 -8385.642,E2 -8385.642} C_VEL
LIN {X 0,Y 452.873,Z 522.189,A -85,B 0,C 180,E1 -8385.964,E2 -8385.964} C_VEL
LIN {X 0,Y 453.088,Z 512.141,A -85,B 0,C 180,E1 -8389.481,E2 -8389.481} C_VEL
LIN {X 0,Y 453.313,Z 504.286,A -85,B 0,C 180,E1 -8392.324,E2 -8392.324} C_VEL
LIN {X 0,Y 453.686,Z 495.372,A -85,B 0,C 180,E1 -8395.706,E2 -8395.706} C_VEL
LIN {X 0,Y 454.089,Z 488.05,A -85,B 0,C 180,E1 -8398.672,E2 -8398.672} C_VEL
LIN {X 0,Y 454.644,Z 481.026,A -85,B 0,C 180,E1 -8401.766,E2 -8401.766} C_VEL
LIN {X 0,Y 455.19,Z 475.881,A -85,B 0,C 180,E1 -8404.302,E2 -8404.302} C_VEL
LIN {X 0,Y 455.42,Z 471.777,A -85,B 0,C 180,E1 -8406.634,E2 -8406.634} C_VEL
LIN {X 0,Y 455.185,Z 469.546,A -85,B 0,C 180,E1 -8408.141,E2 -8408.141} C_VEL
LIN {X 0,Y 454.636,Z 466.415,A -85,B 0,C 180,E1 -8410.758,E2 -8410.758} C_VEL
LIN {X 0,Y 454.227,Z 464.193,A -85,B 0,C 180,E1 -8413.347,E2 -8413.347} C_VEL
LIN {X 0,Y 453.998,Z 462.868,A -85,B 0,C 180,E1 -8415.844,E2 -8415.844} C_VEL
LIN {X 0,Y 453.883,Z 462.305,A -85,B 0,C 180,E1 -8418.255,E2 -8418.255} C_VEL
LIN {X 0,Y 453.832,Z 462.349,A -85,B 0,C 180,E1 -8420.742,E2 -8420.742} C_VEL
LIN {X 0,Y 453.901,Z 463.163,A -85,B 0,C 180,E1 -8423.958,E2 -8423.958} C_VEL
LIN {X 0,Y 453.729,Z 464.652,A -85,B 0,C 180,E1 -8427.171,E2 -8427.171} C_VEL
LIN {X 0,Y 453.517,Z 466.534,A -85,B 0,C 180,E1 -8430.271,E2 -8430.271} C_VEL
LIN {X 0,Y 453.268,Z 468.652,A -85,B 0,C 180,E1 -8433.279,E2 -8433.279} C_VEL
LIN {X 0,Y 453.13,Z 470.925,A -85,B 0,C 180,E1 -8436.218,E2 -8436.218} C_VEL
LIN {X 0,Y 453.021,Z 473.311,A -85,B 0,C 180,E1 -8439.095,E2 -8439.095} C_VEL
LIN {X 0,Y 452.917,Z 475.787,A -85,B 0,C 180,E1 -8441.92,E2 -8441.92} C_VEL
LIN {X 0,Y 452.934,Z 477.86,A -85,B 0,C 180,E1 -8444.192,E2 -8444.192} C_VEL
LIN {X 0,Y 455.997,Z 490.097,A -85,B 0,C 180,E1 -8444.754,E2 -8444.754} C_VEL
LIN {X 0,Y 456.601,Z 493.935,A -85,B 0,C 180,E1 -8444.945,E2 -8444.945} C_VEL
LIN {X 0,Y 456.13,Z 506.666,A -85,B 0,C 180,E1 -8445.614,E2 -8445.614} C_VEL
LIN {X 0,Y 455.678,Z 517.2,A -85,B 0,C 180,E1 -8446.328,E2 -8446.328} C_VEL
LIN {X 0,Y 455.129,Z 528.53,A -85,B 0,C 180,E1 -8447.288,E2 -8447.288} C_VEL
LIN {X 0,Y 454.455,Z 539.081,A -85,B 0,C 180,E1 -8448.402,E2 -8448.402} C_VEL
LIN {X 0,Y 454.071,Z 547.677,A -85,B 0,C 180,E1 -8449.522,E2 -8449.522} C_VEL
LIN {X 0,Y 453.632,Z 556.048,A -85,B 0,C 180,E1 -8450.863,E2 -8450.863} C_VEL
LIN {X 0,Y 453.294,Z 561.762,A -85,B 0,C 180,E1 -8451.979,E2 -8451.979} C_VEL
LIN {X 0,Y 453.033,Z 567.784,A -85,B 0,C 180,E1 -8453.454,E2 -8453.454} C_VEL
LIN {X 0,Y 452.776,Z 572.874,A -85,B 0,C 180,E1 -8455.103,E2 -8455.103} C_VEL
LIN {X 0,Y 452.676,Z 575.795,A -85,B 0,C 180,E1 -8456.44,E2 -8456.44} C_VEL
LIN {X 0,Y 452.652,Z 577.197,A -85,B 0,C 180,E1 -8457.33,E2 -8457.33} C_VEL
LIN {X 0,Y 452.578,Z 578.174,A -85,B 0,C 180,E1 -8458.22,E2 -8458.22} C_VEL
LIN {X 0,Y 452.465,Z 578.964,A -85,B 0,C 180,E1 -8460,E2 -8460} C_VEL
LIN {X 0,Y 452.49,Z 578.725,A -85,B 0,C 180,E1 -8460.89,E2 -8460.89} C_VEL
LIN {X 0,Y 452.577,Z 578.077,A -85,B 0,C 180,E1 -8461.78,E2 -8461.78} C_VEL
LIN {X 0,Y 452.623,Z 577.04,A -85,B 0,C 180,E1 -8462.67,E2 -8462.67} C_VEL
LIN {X 0,Y 452.666,Z 575.601,A -85,B 0,C 180,E1 -8463.561,E2 -8463.561} C_VEL
LIN {X 0,Y 452.703,Z 572.6,A -85,B 0,C 180,E1 -8464.898,E2 -8464.898} C_VEL
LIN {X 0,Y 453.014,Z 567.487,A -85,B 0,C 180,E1 -8466.525,E2 -8466.525} C_VEL
LIN {X 0,Y 453.181,Z 561.277,A -85,B 0,C 180,E1 -8468.023,E2 -8468.023} C_VEL
LIN {X 0,Y 453.554,Z 554.236,A -85,B 0,C 180,E1 -8469.364,E2 -8469.364} C_VEL
LIN {X 0,Y 454.018,Z 545.421,A -85,B 0,C 180,E1 -8470.705,E2 -8470.705} C_VEL
LIN {X 0,Y 454.503,Z 535.436,A -85,B 0,C 180,E1 -8471.936,E2 -8471.936} C_VEL
LIN {X 0,Y 455.033,Z 525.889,A -85,B 0,C 180,E1 -8472.887,E2 -8472.887} C_VEL
LIN {X 0,Y 455.485,Z 514.709,A -85,B 0,C 180,E1 -8473.792,E2 -8473.792} C_VEL
LIN {X 0,Y 455.959,Z 503.597,A -85,B 0,C 180,E1 -8474.506,E2 -8474.506} C_VEL
LIN {X 0,Y 456.273,Z 492.431,A -85,B 0,C 180,E1 -8475.066,E2 -8475.066} C_VEL
LIN {X 0,Y 453.613,Z 479.529,A -85,B 0,C 180,E1 -8475.635,E2 -8475.635} C_VEL
LIN {X 0,Y 452.655,Z 475.465,A -85,B 0,C 180,E1 -8475.81,E2 -8475.81} C_VEL
LIN {X 0,Y 452.644,Z 471.949,A -85,B 0,C 180,E1 -8479.03,E2 -8479.03} C_VEL
LIN {X 0,Y 452.672,Z 468.879,A -85,B 0,C 180,E1 -8481.877,E2 -8481.877} C_VEL
LIN {X 0,Y 452.744,Z 465.801,A -85,B 0,C 180,E1 -8484.78,E2 -8484.78} C_VEL
LIN {X 0,Y 452.816,Z 462.658,A -85,B 0,C 180,E1 -8487.788,E2 -8487.788} C_VEL
LIN {X 0,Y 452.824,Z 460.621,A -85,B 0,C 180,E1 -8489.779,E2 -8489.779} C_VEL
LIN {X 0,Y 452.971,Z 460.065,A -85,B 0,C 180,E1 -8491.422,E2 -8491.422} C_VEL
LIN {X 0,Y 453.358,Z 460.016,A -85,B 0,C 180,E1 -8494.753,E2 -8494.753} C_VEL
LIN {X 0,Y 453.449,Z 460.001,A -85,B 0,C 180,E1 -8497.772,E2 -8497.772} C_VEL
LIN {X 0,Y 453.498,Z 459.996,A -85,B 0,C 180,E1 -8500.609,E2 -8500.609} C_VEL
LIN {X 0,Y 453.468,Z 459.998,A -85,B 0,C 180,E1 -8503.245,E2 -8503.245} C_VEL
LIN {X 0,Y 453.469,Z 460.001,A -85,B 0,C 180,E1 -8505.779,E2 -8505.779} C_VEL
LIN {X 0,Y 453.483,Z 459.997,A -85,B 0,C 180,E1 -8508.209,E2 -8508.209} C_VEL
LIN {X 0,Y 453.52,Z 459.993,A -85,B 0,C 180,E1 -8510.79,E2 -8510.79} C_VEL
LIN {X 0,Y 453.459,Z 460.001,A -85,B 0,C 180,E1 -8513.917,E2 -8513.917} C_VEL
LIN {X 0,Y 453.488,Z 459.996,A -85,B 0,C 180,E1 -8517.151,E2 -8517.151} C_VEL
LIN {X 0,Y 453.48,Z 459.998,A -85,B 0,C 180,E1 -8520.269,E2 -8520.269} C_VEL
LIN {X 0,Y 453.507,Z 459.994,A -85,B 0,C 180,E1 -8523.294,E2 -8523.294} C_VEL
LIN {X 0,Y 453.503,Z 459.997,A -85,B 0,C 180,E1 -8526.239,E2 -8526.239} C_VEL
LIN {X 0,Y 453.488,Z 459.996,A -85,B 0,C 180,E1 -8529.118,E2 -8529.118} C_VEL
LIN {X 0,Y 453.509,Z 459.994,A -85,B 0,C 180,E1 -8531.944,E2 -8531.944} C_VEL
LIN {X 0,Y 453.545,Z 459.99,A -85,B 0,C 180,E1 -8534.726,E2 -8534.726} C_VEL
LIN {X 0,Y 453.565,Z 459.987,A -85,B 0,C 180,E1 -8538.379,E2 -8538.379} C_VEL
LIN {X 0,Y 453.532,Z 459.988,A -85,B 0,C 180,E1 -8539.089,E2 -8539.089} C_VEL
LIN {X 0,Y 452.882,Z 460.074,A -85,B 0,C 180,E1 -8539.831,E2 -8539.831} C_VEL
LIN {X 0,Y 450.074,Z 460.422,A -85,B 0,C 180,E1 -8541.036,E2 -8541.036} C_VEL
LIN {X 0,Y 447.7,Z 460.719,A -85,B 0,C 180,E1 -8542.008,E2 -8542.008} C_VEL
LIN {X 0,Y 446.691,Z 460.844,A -85,B 0,C 180,E1 -8542.759,E2 -8542.759} C_VEL
LIN {X 0,Y 446.614,Z 460.852,A -85,B 0,C 180,E1 -8543.013,E2 -8543.013} C_VEL
LIN {X 0,Y 446.65,Z 460.85,A -85,B 0,C 180,E1 -8544.583,E2 -8544.583} C_VEL
LIN {X 0,Y 446.67,Z 460.848,A -85,B 0,C 180,E1 -8548.197,E2 -8548.197} C_VEL
LIN {X 0,Y 446.799,Z 460.832,A -85,B 0,C 180,E1 -8550,E2 -8550} C_VEL
LIN {X 0,Y 446.696,Z 460.841,A -85,B 0,C 180,E1 -8552.705,E2 -8552.705} C_VEL
LIN {X 0,Y 446.625,Z 460.852,A -85,B 0,C 180,E1 -8556.324,E2 -8556.324} C_VEL
LIN {X 0,Y 446.527,Z 460.864,A -85,B 0,C 180,E1 -8559.97,E2 -8559.97} C_VEL
LIN {X 0,Y 446.527,Z 460.862,A -85,B 0,C 180,E1 -8562.73,E2 -8562.73} C_VEL
LIN {X 0,Y 446.502,Z 460.866,A -85,B 0,C 180,E1 -8566.228,E2 -8566.228} C_VEL
LIN {X 0,Y 446.475,Z 460.872,A -85,B 0,C 180,E1 -8569.303,E2 -8569.303} C_VEL
LIN {X 0,Y 446.424,Z 460.879,A -85,B 0,C 180,E1 -8572.199,E2 -8572.199} C_VEL
LIN {X 0,Y 446.449,Z 460.871,A -85,B 0,C 180,E1 -8575.153,E2 -8575.153} C_VEL
LIN {X 0,Y 446.49,Z 460.868,A -85,B 0,C 180,E1 -8578.178,E2 -8578.178} C_VEL
LIN {X 0,Y 446.424,Z 460.877,A -85,B 0,C 180,E1 -8581.775,E2 -8581.775} C_VEL
LIN {X 0,Y 446.435,Z 460.876,A -85,B 0,C 180,E1 -8584.523,E2 -8584.523} C_VEL
LIN {X 0,Y 446.435,Z 460.876,A -85,B 0,C 180,E1 -8588.082,E2 -8588.082} C_VEL
LIN {X 0,Y 446.431,Z 460.874,A -85,B 0,C 180,E1 -8590.917,E2 -8590.917} C_VEL
LIN {X 0,Y 446.406,Z 460.879,A -85,B 0,C 180,E1 -8593.846,E2 -8593.846} C_VEL
LIN {X 0,Y 446.425,Z 460.877,A -85,B 0,C 180,E1 -8596.4,E2 -8596.4} C_VEL
LIN {X 0,Y 446.448,Z 460.876,A -85,B 0,C 180,E1 -8599.802,E2 -8599.802} C_VEL
LIN {X 0,Y 446.395,Z 460.881,A -85,B 0,C 180,E1 -8603.254,E2 -8603.254} C_VEL
LIN {X 0,Y 446.318,Z 460.892,A -85,B 0,C 180,E1 -8605.467,E2 -8605.467} C_VEL
LIN {X 0,Y 446.029,Z 460.928,A -85,B 0,C 180,E1 -8608.307,E2 -8608.307} C_VEL
LIN {X 0,Y 445.678,Z 460.974,A -85,B 0,C 180,E1 -8610.735,E2 -8610.735} C_VEL
LIN {X 0,Y 445.666,Z 461.829,A -85,B 0,C 180,E1 -8612.019,E2 -8612.019} C_VEL
LIN {X 0,Y 445.605,Z 464.982,A -85,B 0,C 180,E1 -8614.796,E2 -8614.796} C_VEL
LIN {X 0,Y 445.556,Z 468.37,A -85,B 0,C 180,E1 -8617.755,E2 -8617.755} C_VEL
LIN {X 0,Y 445.55,Z 472.235,A -85,B 0,C 180,E1 -8621.161,E2 -8621.161} C_VEL
LIN {X 0,Y 445.531,Z 475.647,A -85,B 0,C 180,E1 -8624.104,E2 -8624.104} C_VEL
LIN {X 0,Y 448.418,Z 488.597,A -85,B 0,C 180,E1 -8624.627,E2 -8624.627} C_VEL
LIN {X 0,Y 449.353,Z 493.523,A -85,B 0,C 180,E1 -8624.87,E2 -8624.87} C_VEL
LIN {X 0,Y 448.914,Z 505.42,A -85,B 0,C 180,E1 -8625.493,E2 -8625.493} C_VEL
LIN {X 0,Y 448.444,Z 517.624,A -85,B 0,C 180,E1 -8626.328,E2 -8626.328} C_VEL
LIN {X 0,Y 447.936,Z 528.926,A -85,B 0,C 180,E1 -8627.311,E2 -8627.311} C_VEL
LIN {X 0,Y 447.264,Z 539.379,A -85,B 0,C 180,E1 -8628.443,E2 -8628.443} C_VEL
LIN {X 0,Y 446.835,Z 547.947,A -85,B 0,C 180,E1 -8629.579,E2 -8629.579} C_VEL
LIN {X 0,Y 446.402,Z 556.291,A -85,B 0,C 180,E1 -8630.942,E2 -8630.942} C_VEL
LIN {X 0,Y 446.027,Z 562.997,A -85,B 0,C 180,E1 -8632.303,E2 -8632.303} C_VEL
LIN {X 0,Y 445.908,Z 568.349,A -85,B 0,C 180,E1 -8633.666,E2 -8633.666} C_VEL
LIN {X 0,Y 445.605,Z 572.526,A -85,B 0,C 180,E1 -8635.023,E2 -8635.023} C_VEL
LIN {X 0,Y 445.608,Z 575.623,A -85,B 0,C 180,E1 -8636.383,E2 -8636.383} C_VEL
LIN {X 0,Y 445.536,Z 577.161,A -85,B 0,C 180,E1 -8637.287,E2 -8637.287} C_VEL
LIN {X 0,Y 445.488,Z 578.239,A -85,B 0,C 180,E1 -8638.192,E2 -8638.192} C_VEL
LIN {X 0,Y 445.401,Z 579.229,A -85,B 0,C 180,E1 -8640,E2 -8640} C_VEL
LIN {X 0,Y 445.428,Z 579.093,A -85,B 0,C 180,E1 -8640.904,E2 -8640.904} C_VEL
LIN {X 0,Y 445.521,Z 578.541,A -85,B 0,C 180,E1 -8641.808,E2 -8641.808} C_VEL
LIN {X 0,Y 445.572,Z 577.605,A -85,B 0,C 180,E1 -8642.712,E2 -8642.712} C_VEL
LIN {X 0,Y 445.62,Z 576.26,A -85,B 0,C 180,E1 -8643.617,E2 -8643.617} C_VEL
LIN {X 0,Y 445.677,Z 573.409,A -85,B 0,C 180,E1 -8644.975,E2 -8644.975} C_VEL
LIN {X 0,Y 445.936,Z 569.495,A -85,B 0,C 180,E1 -8646.334,E2 -8646.334} C_VEL
LIN {X 0,Y 446.128,Z 564.416,A -85,B 0,C 180,E1 -8647.695,E2 -8647.695} C_VEL
LIN {X 0,Y 446.592,Z 556.808,A -85,B 0,C 180,E1 -8649.282,E2 -8649.282} C_VEL
LIN {X 0,Y 447.033,Z 548.542,A -85,B 0,C 180,E1 -8650.645,E2 -8650.645} C_VEL
LIN {X 0,Y 447.461,Z 540.107,A -85,B 0,C 180,E1 -8651.782,E2 -8651.782} C_VEL
LIN {X 0,Y 448.155,Z 529.947,A -85,B 0,C 180,E1 -8652.897,E2 -8652.897} C_VEL
LIN {X 0,Y 448.701,Z 518.335,A -85,B 0,C 180,E1 -8653.916,E2 -8653.916} C_VEL
LIN {X 0,Y 449.311,Z 506.649,A -85,B 0,C 180,E1 -8654.725,E2 -8654.725} C_VEL
LIN {X 0,Y 449.787,Z 494.987,A -85,B 0,C 180,E1 -8655.346,E2 -8655.346} C_VEL
LIN {X 0,Y 447.794,Z 485.131,A -85,B 0,C 180,E1 -8655.848,E2 -8655.848} C_VEL
LIN {X 0,Y 445.74,Z 477.69,A -85,B 0,C 180,E1 -8656.194,E2 -8656.194} C_VEL
LIN {X 0,Y 445.749,Z 474.111,A -85,B 0,C 180,E1 -8659.336,E2 -8659.336} C_VEL
LIN {X 0,Y 445.749,Z 470.751,A -85,B 0,C 180,E1 -8662.235,E2 -8662.235} C_VEL
LIN {X 0,Y 445.793,Z 467.272,A -85,B 0,C 180,E1 -8665.192,E2 -8665.192} C_VEL
LIN {X 0,Y 445.801,Z 463.489,A -85,B 0,C 180,E1 -8668.226,E2 -8668.226} C_VEL
LIN {X 0,Y 445.78,Z 460.961,A -85,B 0,C 180,E1 -8670.298,E2 -8670.298} C_VEL
LIN {X 0,Y 446.117,Z 460.919,A -85,B 0,C 180,E1 -8672.386,E2 -8672.386} C_VEL
LIN {X 0,Y 446.354,Z 460.887,A -85,B 0,C 180,E1 -8675.039,E2 -8675.039} C_VEL
LIN {X 0,Y 446.417,Z 460.879,A -85,B 0,C 180,E1 -8678.079,E2 -8678.079} C_VEL
LIN {X 0,Y 446.43,Z 460.879,A -85,B 0,C 180,E1 -8680.918,E2 -8680.918} C_VEL
LIN {X 0,Y 446.425,Z 460.878,A -85,B 0,C 180,E1 -8683.843,E2 -8683.843} C_VEL
LIN {X 0,Y 446.402,Z 460.881,A -85,B 0,C 180,E1 -8686.403,E2 -8686.403} C_VEL
LIN {X 0,Y 446.484,Z 460.986,A -85,B 0,C 180,E1 -8688.68,E2 -8688.68} C_VEL
LIN {X 0,Y 447.64,Z 467.448,A -85,B 0,C 180,E1 -8691.721,E2 -8691.721} C_VEL
LIN {X 0,Y 448.366,Z 472.51,A -85,B 0,C 180,E1 -8693.999,E2 -8693.999} C_VEL
LIN {X 0,Y 447.986,Z 478.942,A -85,B 0,C 180,E1 -8696.696,E2 -8696.696} C_VEL
LIN {X 0,Y 447.469,Z 486.656,A -85,B 0,C 180,E1 -8699.828,E2 -8699.828} C_VEL
LIN {X 0,Y 447.018,Z 494.379,A -85,B 0,C 180,E1 -8702.875,E2 -8702.875} C_VEL
LIN {X 0,Y 446.618,Z 502.203,A -85,B 0,C 180,E1 -8705.88,E2 -8705.88} C_VEL
LIN {X 0,Y 446.286,Z 509.873,A -85,B 0,C 180,E1 -8708.765,E2 -8708.765} C_VEL
LIN {X 0,Y 445.964,Z 518.915,A -85,B 0,C 180,E1 -8712.103,E2 -8712.103} C_VEL
LIN {X 0,Y 445.878,Z 523.911,A -85,B 0,C 180,E1 -8713.925,E2 -8713.925} C_VEL
LIN {X 0,Y 447.933,Z 538.631,A -85,B 0,C 180,E1 -8714.45,E2 -8714.45} C_VEL
LIN {X 0,Y 448.974,Z 548.521,A -85,B 0,C 180,E1 -8714.916,E2 -8714.916} C_VEL
LIN {X 0,Y 448.418,Z 560.539,A -85,B 0,C 180,E1 -8715.593,E2 -8715.593} C_VEL
LIN {X 0,Y 447.822,Z 572.681,A -85,B 0,C 180,E1 -8716.48,E2 -8716.48} C_VEL
LIN {X 0,Y 447.231,Z 583.938,A -85,B 0,C 180,E1 -8717.521,E2 -8717.521} C_VEL
LIN {X 0,Y 446.705,Z 593.811,A -85,B 0,C 180,E1 -8718.658,E2 -8718.658} C_VEL
LIN {X 0,Y 446.172,Z 603.413,A -85,B 0,C 180,E1 -8720.022,E2 -8720.022} C_VEL
LIN {X 0,Y 445.874,Z 611.069,A -85,B 0,C 180,E1 -8721.388,E2 -8721.388} C_VEL
LIN {X 0,Y 445.615,Z 617.223,A -85,B 0,C 180,E1 -8722.752,E2 -8722.752} C_VEL
LIN {X 0,Y 445.494,Z 621.498,A -85,B 0,C 180,E1 -8723.927,E2 -8723.927} C_VEL
LIN {X 0,Y 445.43,Z 625.817,A -85,B 0,C 180,E1 -8725.475,E2 -8725.475} C_VEL
LIN {X 0,Y 445.428,Z 627.732,A -85,B 0,C 180,E1 -8726.382,E2 -8726.382} C_VEL
LIN {X 0,Y 445.467,Z 629.181,A -85,B 0,C 180,E1 -8727.287,E2 -8727.287} C_VEL
LIN {X 0,Y 445.45,Z 630.189,A -85,B 0,C 180,E1 -8728.192,E2 -8728.192} C_VEL
LIN {X 0,Y 445.426,Z 630.793,A -85,B 0,C 180,E1 -8729.096,E2 -8729.096} C_VEL
LIN {X 0,Y 445.399,Z 630.994,A -85,B 0,C 180,E1 -8730,E2 -8730} C_VEL
LIN {X 0,Y 445.427,Z 630.75,A -85,B 0,C 180,E1 -8730.904,E2 -8730.904} C_VEL
LIN {X 0,Y 445.452,Z 630.087,A -85,B 0,C 180,E1 -8731.808,E2 -8731.808} C_VEL
LIN {X 0,Y 445.475,Z 629.021,A -85,B 0,C 180,E1 -8732.713,E2 -8732.713} C_VEL
LIN {X 0,Y 445.441,Z 627.534,A -85,B 0,C 180,E1 -8733.618,E2 -8733.618} C_VEL
LIN {X 0,Y 445.492,Z 624.436,A -85,B 0,C 180,E1 -8734.978,E2 -8734.978} C_VEL
LIN {X 0,Y 445.529,Z 620.095,A -85,B 0,C 180,E1 -8736.386,E2 -8736.386} C_VEL
LIN {X 0,Y 445.719,Z 613.844,A -85,B 0,C 180,E1 -8737.93,E2 -8737.93} C_VEL
LIN {X 0,Y 446.023,Z 606.882,A -85,B 0,C 180,E1 -8739.295,E2 -8739.295} C_VEL
LIN {X 0,Y 446.378,Z 598.277,A -85,B 0,C 180,E1 -8740.661,E2 -8740.661} C_VEL
LIN {X 0,Y 446.944,Z 589.466,A -85,B 0,C 180,E1 -8741.796,E2 -8741.796} C_VEL
LIN {X 0,Y 447.329,Z 581.058,A -85,B 0,C 180,E1 -8742.706,E2 -8742.706} C_VEL
LIN {X 0,Y 447.92,Z 569.588,A -85,B 0,C 180,E1 -8743.728,E2 -8743.728} C_VEL
LIN {X 0,Y 448.515,Z 558.526,A -85,B 0,C 180,E1 -8744.52,E2 -8744.52} C_VEL
LIN {X 0,Y 448.944,Z 546.478,A -85,B 0,C 180,E1 -8745.201,E2 -8745.201} C_VEL
LIN {X 0,Y 447.343,Z 531.722,A -85,B 0,C 180,E1 -8745.89,E2 -8745.89} C_VEL
LIN {X 0,Y 445.803,Z 521.639,A -85,B 0,C 180,E1 -8746.273,E2 -8746.273} C_VEL
LIN {X 0,Y 446.039,Z 511.804,A -85,B 0,C 180,E1 -8749.802,E2 -8749.802} C_VEL
LIN {X 0,Y 446.276,Z 504.023,A -85,B 0,C 180,E1 -8752.695,E2 -8752.695} C_VEL
LIN {X 0,Y 446.71,Z 494.897,A -85,B 0,C 180,E1 -8756.263,E2 -8756.263} C_VEL
LIN {X 0,Y 447.141,Z 488.006,A -85,B 0,C 180,E1 -8759.16,E2 -8759.16} C_VEL
LIN {X 0,Y 447.734,Z 481.259,A -85,B 0,C 180,E1 -8762.255,E2 -8762.255} C_VEL
LIN {X 0,Y 448.244,Z 477.12,A -85,B 0,C 180,E1 -8764.364,E2 -8764.364} C_VEL
LIN {X 0,Y 448.435,Z 472.774,A -85,B 0,C 180,E1 -8766.938,E2 -8766.938} C_VEL
LIN {X 0,Y 448.083,Z 470.124,A -85,B 0,C 180,E1 -8768.858,E2 -8768.858} C_VEL
LIN {X 0,Y 447.607,Z 467.475,A -85,B 0,C 180,E1 -8771.258,E2 -8771.258} C_VEL
LIN {X 0,Y 447.236,Z 465.499,A -85,B 0,C 180,E1 -8773.744,E2 -8773.744} C_VEL
LIN {X 0,Y 447.038,Z 464.239,A -85,B 0,C 180,E1 -8776.318,E2 -8776.318} C_VEL
LIN {X 0,Y 446.917,Z 463.727,A -85,B 0,C 180,E1 -8779.01,E2 -8779.01} C_VEL
LIN {X 0,Y 446.914,Z 463.993,A -85,B 0,C 180,E1 -8782.172,E2 -8782.172} C_VEL
LIN {X 0,Y 446.878,Z 464.806,A -85,B 0,C 180,E1 -8784.865,E2 -8784.865} C_VEL
LIN {X 0,Y 446.676,Z 466.128,A -85,B 0,C 180,E1 -8787.659,E2 -8787.659} C_VEL
LIN {X 0,Y 446.439,Z 468.005,A -85,B 0,C 180,E1 -8790.79,E2 -8790.79} C_VEL
LIN {X 0,Y 446.227,Z 470.124,A -85,B 0,C 180,E1 -8793.863,E2 -8793.863} C_VEL
LIN {X 0,Y 446.05,Z 472.375,A -85,B 0,C 180,E1 -8796.803,E2 -8796.803} C_VEL
LIN {X 0,Y 445.922,Z 474.764,A -85,B 0,C 180,E1 -8799.712,E2 -8799.712} C_VEL
LIN {X 0,Y 445.848,Z 477.249,A -85,B 0,C 180,E1 -8802.572,E2 -8802.572} C_VEL
LIN {X 0,Y 445.882,Z 478.544,A -85,B 0,C 180,E1 -8803.894,E2 -8803.894} C_VEL
LIN {X 0,Y 449.062,Z 490.483,A -85,B 0,C 180,E1 -8804.475,E2 -8804.475} C_VEL
LIN {X 0,Y 449.823,Z 495.06,A -85,B 0,C 180,E1 -8804.713,E2 -8804.713} C_VEL
LIN {X 0,Y 449.321,Z 507.604,A -85,B 0,C 180,E1 -8805.391,E2 -8805.391} C_VEL
LIN {X 0,Y 448.852,Z 518.031,A -85,B 0,C 180,E1 -8806.116,E2 -8806.116} C_VEL
LIN {X 0,Y 448.242,Z 529.25,A -85,B 0,C 180,E1 -8807.09,E2 -8807.09} C_VEL
LIN {X 0,Y 447.53,Z 539.704,A -85,B 0,C 180,E1 -8808.22,E2 -8808.22} C_VEL
LIN {X 0,Y 447.115,Z 548.229,A -85,B 0,C 180,E1 -8809.357,E2 -8809.357} C_VEL
LIN {X 0,Y 446.651,Z 556.56,A -85,B 0,C 180,E1 -8810.719,E2 -8810.719} C_VEL
LIN {X 0,Y 446.267,Z 562.268,A -85,B 0,C 180,E1 -8811.852,E2 -8811.852} C_VEL
LIN {X 0,Y 445.998,Z 567.404,A -85,B 0,C 180,E1 -8813.099,E2 -8813.099} C_VEL
LIN {X 0,Y 445.662,Z 572.148,A -85,B 0,C 180,E1 -8814.571,E2 -8814.571} C_VEL
LIN {X 0,Y 445.765,Z 574.413,A -85,B 0,C 180,E1 -8815.479,E2 -8815.479} C_VEL
LIN {X 0,Y 445.62,Z 576.267,A -85,B 0,C 180,E1 -8816.383,E2 -8816.383} C_VEL
LIN {X 0,Y 445.572,Z 577.656,A -85,B 0,C 180,E1 -8817.288,E2 -8817.288} C_VEL
LIN {X 0,Y 445.521,Z 578.623,A -85,B 0,C 180,E1 -8818.192,E2 -8818.192} C_VEL
LIN {X 0,Y 445.401,Z 579.386,A -85,B 0,C 180,E1 -8820,E2 -8820} C_VEL
LIN {X 0,Y 445.428,Z 579.128,A -85,B 0,C 180,E1 -8820.904,E2 -8820.904} C_VEL
LIN {X 0,Y 445.502,Z 578.469,A -85,B 0,C 180,E1 -8821.808,E2 -8821.808} C_VEL
LIN {X 0,Y 445.546,Z 577.421,A -85,B 0,C 180,E1 -8822.713,E2 -8822.713} C_VEL
LIN {X 0,Y 445.608,Z 575.96,A -85,B 0,C 180,E1 -8823.617,E2 -8823.617} C_VEL
LIN {X 0,Y 445.622,Z 572.935,A -85,B 0,C 180,E1 -8824.976,E2 -8824.976} C_VEL
LIN {X 0,Y 445.91,Z 568.843,A -85,B 0,C 180,E1 -8826.334,E2 -8826.334} C_VEL
LIN {X 0,Y 446.089,Z 562.56,A -85,B 0,C 180,E1 -8827.924,E2 -8827.924} C_VEL
LIN {X 0,Y 446.47,Z 555.719,A -85,B 0,C 180,E1 -8829.285,E2 -8829.285} C_VEL
LIN {X 0,Y 446.939,Z 547.213,A -85,B 0,C 180,E1 -8830.648,E2 -8830.648} C_VEL
LIN {X 0,Y 447.354,Z 538.472,A -85,B 0,C 180,E1 -8831.785,E2 -8831.785} C_VEL
LIN {X 0,Y 447.981,Z 528.197,A -85,B 0,C 180,E1 -8832.875,E2 -8832.875} C_VEL
LIN {X 0,Y 448.426,Z 517.696,A -85,B 0,C 180,E1 -8833.784,E2 -8833.784} C_VEL
LIN {X 0,Y 448.985,Z 505.388,A -85,B 0,C 180,E1 -8834.62,E2 -8834.62} C_VEL
LIN {X 0,Y 449.361,Z 493.421,A -85,B 0,C 180,E1 -8835.245,E2 -8835.245} C_VEL
LIN {X 0,Y 446.618,Z 480.351,A -85,B 0,C 180,E1 -8835.84,E2 -8835.84} C_VEL
LIN {X 0,Y 445.56,Z 475.833,A -85,B 0,C 180,E1 -8836.015,E2 -8836.015} C_VEL
LIN {X 0,Y 445.574,Z 472.212,A -85,B 0,C 180,E1 -8839.344,E2 -8839.344} C_VEL
LIN {X 0,Y 445.584,Z 469.11,A -85,B 0,C 180,E1 -8842.244,E2 -8842.244} C_VEL
LIN {X 0,Y 445.68,Z 465.996,A -85,B 0,C 180,E1 -8845.2,E2 -8845.2} C_VEL
LIN {X 0,Y 445.757,Z 462.865,A -85,B 0,C 180,E1 -8848.229,E2 -8848.229} C_VEL
LIN {X 0,Y 445.774,Z 460.966,A -85,B 0,C 180,E1 -8850.299,E2 -8850.299} C_VEL
LIN {X 0,Y 446.153,Z 460.912,A -85,B 0,C 180,E1 -8853.459,E2 -8853.459} C_VEL
LIN {X 0,Y 446.347,Z 460.887,A -85,B 0,C 180,E1 -8855.633,E2 -8855.633} C_VEL
LIN {X 0,Y 446.441,Z 460.873,A -85,B 0,C 180,E1 -8859.028,E2 -8859.028} C_VEL
LIN {X 0,Y 446.441,Z 460.877,A -85,B 0,C 180,E1 -8862.278,E2 -8862.278} C_VEL
LIN {X 0,Y 446.459,Z 460.872,A -85,B 0,C 180,E1 -8865.103,E2 -8865.103} C_VEL
LIN {X 0,Y 446.432,Z 460.877,A -85,B 0,C 180,E1 -8868.609,E2 -8868.609} C_VEL
LIN {X 0,Y 446.465,Z 460.871,A -85,B 0,C 180,E1 -8870.975,E2 -8870.975} C_VEL
LIN {X 0,Y 446.424,Z 460.878,A -85,B 0,C 180,E1 -8874.374,E2 -8874.374} C_VEL
LIN {X 0,Y 446.427,Z 460.877,A -85,B 0,C 180,E1 -8877.639,E2 -8877.639} C_VEL
LIN {X 0,Y 446.454,Z 460.874,A -85,B 0,C 180,E1 -8880.791,E2 -8880.791} C_VEL
LIN {X 0,Y 446.483,Z 460.869,A -85,B 0,C 180,E1 -8883.849,E2 -8883.849} C_VEL
LIN {X 0,Y 446.432,Z 460.873,A -85,B 0,C 180,E1 -8886.823,E2 -8886.823} C_VEL
LIN {X 0,Y 446.449,Z 460.876,A -85,B 0,C 180,E1 -8889.737,E2 -8889.737} C_VEL
LIN {X 0,Y 446.463,Z 460.873,A -85,B 0,C 180,E1 -8892.597,E2 -8892.597} C_VEL
LIN {X 0,Y 446.476,Z 460.87,A -85,B 0,C 180,E1 -8895.413,E2 -8895.413} C_VEL
LIN {X 0,Y 446.523,Z 460.867,A -85,B 0,C 180,E1 -8898.193,E2 -8898.193} C_VEL
LIN {X 0,Y 446.606,Z 460.856,A -85,B 0,C 180,E1 -8901.858,E2 -8901.858} C_VEL
LIN {X 0,Y 446.614,Z 460.852,A -85,B 0,C 180,E1 -8903.013,E2 -8903.013} C_VEL
LIN {X 0,Y 445.928,Z 460.94,A -85,B 0,C 180,E1 -8903.765,E2 -8903.765} C_VEL
LIN {X 0,Y 442.974,Z 461.306,A -85,B 0,C 180,E1 -8904.985,E2 -8904.985} C_VEL
LIN {X 0,Y 440.542,Z 461.609,A -85,B 0,C 180,E1 -8905.97,E2 -8905.97} C_VEL
LIN {X 0,Y 439.597,Z 461.727,A -85,B 0,C 180,E1 -8906.732,E2 -8906.732} C_VEL
LIN {X 0,Y 439.573,Z 461.729,A -85,B 0,C 180,E1 -8906.99,E2 -8906.99} C_VEL
LIN {X 0,Y 439.768,Z 461.708,A -85,B 0,C 180,E1 -8910,E2 -8910} C_VEL
LIN {X 0,Y 439.646,Z 461.719,A -85,B 0,C 180,E1 -8912.749,E2 -8912.749} C_VEL
LIN {X 0,Y 439.597,Z 461.727,A -85,B 0,C 180,E1 -8916.426,E2 -8916.426} C_VEL
LIN {X 0,Y 439.501,Z 461.739,A -85,B 0,C 180,E1 -8919.202,E2 -8919.202} C_VEL
LIN {X 0,Y 439.471,Z 461.74,A -85,B 0,C 180,E1 -8922.938,E2 -8922.938} C_VEL
LIN {X 0,Y 439.453,Z 461.744,A -85,B 0,C 180,E1 -8926.349,E2 -8926.349} C_VEL
LIN {X 0,Y 439.408,Z 461.751,A -85,B 0,C 180,E1 -8929.626,E2 -8929.626} C_VEL
LIN {X 0,Y 439.369,Z 461.755,A -85,B 0,C 180,E1 -8932.575,E2 -8932.575} C_VEL
LIN {X 0,Y 439.403,Z 461.751,A -85,B 0,C 180,E1 -8935.585,E2 -8935.585} C_VEL
LIN {X 0,Y 439.422,Z 461.748,A -85,B 0,C 180,E1 -8938.673,E2 -8938.673} C_VEL
LIN {X 0,Y 439.375,Z 461.755,A -85,B 0,C 180,E1 -8942.03,E2 -8942.03} C_VEL
LIN {X 0,Y 439.401,Z 461.751,A -85,B 0,C 180,E1 -8945.341,E2 -8945.341} C_VEL
LIN {X 0,Y 439.395,Z 461.749,A -85,B 0,C 180,E1 -8948.594,E2 -8948.594} C_VEL
LIN {X 0,Y 439.393,Z 461.753,A -85,B 0,C 180,E1 -8951.257,E2 -8951.257} C_VEL
LIN {X 0,Y 439.407,Z 461.751,A -85,B 0,C 180,E1 -8954.729,E2 -8954.729} C_VEL
LIN {X 0,Y 439.402,Z 461.752,A -85,B 0,C 180,E1 -8957.796,E2 -8957.796} C_VEL
LIN {X 0,Y 439.43,Z 461.747,A -85,B 0,C 180,E1 -8960.227,E2 -8960.227} C_VEL
LIN {X 0,Y 439.355,Z 461.759,A -85,B 0,C 180,E1 -8963.711,E2 -8963.711} C_VEL
LIN {X 0,Y 439.235,Z 461.773,A -85,B 0,C 180,E1 -8966.308,E2 -8966.308} C_VEL
LIN {X 0,Y 438.838,Z 461.824,A -85,B 0,C 180,E1 -8969.17,E2 -8969.17} C_VEL
LIN {X 0,Y 438.595,Z 461.857,A -85,B 0,C 180,E1 -8971.267,E2 -8971.267} C_VEL
LIN {X 0,Y 438.567,Z 463.952,A -85,B 0,C 180,E1 -8973.339,E2 -8973.339} C_VEL
LIN {X 0,Y 438.51,Z 467.379,A -85,B 0,C 180,E1 -8976.379,E2 -8976.379} C_VEL
LIN {X 0,Y 438.468,Z 470.762,A -85,B 0,C 180,E1 -8979.351,E2 -8979.351} C_VEL
LIN {X 0,Y 438.425,Z 474.097,A -85,B 0,C 180,E1 -8982.267,E2 -8982.267} C_VEL
LIN {X 0,Y 438.473,Z 475.918,A -85,B 0,C 180,E1 -8983.866,E2 -8983.866} C_VEL
LIN {X 0,Y 441.407,Z 489.16,A -85,B 0,C 180,E1 -8984.422,E2 -8984.422} C_VEL
LIN {X 0,Y 442.412,Z 495.531,A -85,B 0,C 180,E1 -8984.745,E2 -8984.745} C_VEL
LIN {X 0,Y 441.875,Z 508.848,A -85,B 0,C 180,E1 -8985.492,E2 -8985.492} C_VEL
LIN {X 0,Y 441.394,Z 520.478,A -85,B 0,C 180,E1 -8986.35,E2 -8986.35} C_VEL
LIN {X 0,Y 440.79,Z 532.293,A -85,B 0,C 180,E1 -8987.453,E2 -8987.453} C_VEL
LIN {X 0,Y 440.201,Z 541.304,A -85,B 0,C 180,E1 -8988.488,E2 -8988.488} C_VEL
LIN {X 0,Y 439.658,Z 551.041,A -85,B 0,C 180,E1 -8989.872,E2 -8989.872} C_VEL
LIN {X 0,Y 439.223,Z 558.898,A -85,B 0,C 180,E1 -8991.256,E2 -8991.256} C_VEL
LIN {X 0,Y 438.917,Z 565.161,A -85,B 0,C 180,E1 -8992.64,E2 -8992.64} C_VEL
LIN {X 0,Y 438.761,Z 570.135,A -85,B 0,C 180,E1 -8994.024,E2 -8994.024} C_VEL
LIN {X 0,Y 438.554,Z 573.976,A -85,B 0,C 180,E1 -8995.404,E2 -8995.404} C_VEL
LIN {X 0,Y 438.549,Z 575.955,A -85,B 0,C 180,E1 -8996.324,E2 -8996.324} C_VEL
LIN {X 0,Y 438.464,Z 577.517,A -85,B 0,C 180,E1 -8997.244,E2 -8997.244} C_VEL
LIN {X 0,Y 438.403,Z 578.614,A -85,B 0,C 180,E1 -8998.162,E2 -8998.162} C_VEL
LIN {X 0,Y 438.339,Z 579.631,A -85,B 0,C 180,E1 -9000,E2 -9000} C_VEL
LIN {X 0,Y 438.368,Z 579.514,A -85,B 0,C 180,E1 -9000.918,E2 -9000.918} C_VEL
LIN {X 0,Y 438.465,Z 578.973,A -85,B 0,C 180,E1 -9001.837,E2 -9001.837} C_VEL
LIN {X 0,Y 438.497,Z 578.047,A -85,B 0,C 180,E1 -9002.756,E2 -9002.756} C_VEL
LIN {X 0,Y 438.566,Z 576.712,A -85,B 0,C 180,E1 -9003.675,E2 -9003.675} C_VEL
LIN {X 0,Y 438.621,Z 573.872,A -85,B 0,C 180,E1 -9005.056,E2 -9005.056} C_VEL
LIN {X 0,Y 438.897,Z 569.974,A -85,B 0,C 180,E1 -9006.436,E2 -9006.436} C_VEL
LIN {X 0,Y 439.101,Z 564.93,A -85,B 0,C 180,E1 -9007.819,E2 -9007.819} C_VEL
LIN {X 0,Y 439.597,Z 557.373,A -85,B 0,C 180,E1 -9009.431,E2 -9009.431} C_VEL
LIN {X 0,Y 440.088,Z 549.161,A -85,B 0,C 180,E1 -9010.815,E2 -9010.815} C_VEL
LIN {X 0,Y 440.543,Z 540.754,A -85,B 0,C 180,E1 -9011.969,E2 -9011.969} C_VEL
LIN {X 0,Y 441.264,Z 530.732,A -85,B 0,C 180,E1 -9013.091,E2 -9013.091} C_VEL
LIN {X 0,Y 441.854,Z 519.169,A -85,B 0,C 180,E1 -9014.131,E2 -9014.131} C_VEL
LIN {X 0,Y 442.513,Z 507.565,A -85,B 0,C 180,E1 -9014.956,E2 -9014.956} C_VEL
LIN {X 0,Y 442.947,Z 495.016,A -85,B 0,C 180,E1 -9015.648,E2 -9015.648} C_VEL
LIN {X 0,Y 440.459,Z 484.345,A -85,B 0,C 180,E1 -9016.22,E2 -9016.22} C_VEL
LIN {X 0,Y 438.66,Z 478.19,A -85,B 0,C 180,E1 -9016.521,E2 -9016.521} C_VEL
LIN {X 0,Y 438.697,Z 474.638,A -85,B 0,C 180,E1 -9019.659,E2 -9019.659} C_VEL
LIN {X 0,Y 438.704,Z 471.259,A -85,B 0,C 180,E1 -9022.611,E2 -9022.611} C_VEL
LIN {X 0,Y 438.76,Z 467.63,A -85,B 0,C 180,E1 -9025.625,E2 -9025.625} C_VEL
LIN {X 0,Y 438.749,Z 463.939,A -85,B 0,C 180,E1 -9028.721,E2 -9028.721} C_VEL
LIN {X 0,Y 438.759,Z 462.173,A -85,B 0,C 180,E1 -9030.121,E2 -9030.121} C_VEL
LIN {X 0,Y 439.005,Z 461.805,A -85,B 0,C 180,E1 -9031.89,E2 -9031.89} C_VEL
LIN {X 0,Y 439.232,Z 461.776,A -85,B 0,C 180,E1 -9034.057,E2 -9034.057} C_VEL
LIN {X 0,Y 439.346,Z 461.761,A -85,B 0,C 180,E1 -9036.886,E2 -9036.886} C_VEL
LIN {X 0,Y 439.415,Z 461.751,A -85,B 0,C 180,E1 -9039.851,E2 -9039.851} C_VEL
LIN {X 0,Y 439.388,Z 461.755,A -85,B 0,C 180,E1 -9042.627,E2 -9042.627} C_VEL
LIN {X 0,Y 439.404,Z 461.753,A -85,B 0,C 180,E1 -9045.271,E2 -9045.271} C_VEL
LIN {X 0,Y 439.43,Z 461.885,A -85,B 0,C 180,E1 -9048.428,E2 -9048.428} C_VEL
LIN {X 0,Y 440.597,Z 468.351,A -85,B 0,C 180,E1 -9051.531,E2 -9051.531} C_VEL
LIN {X 0,Y 441.351,Z 473.535,A -85,B 0,C 180,E1 -9053.901,E2 -9053.901} C_VEL
LIN {X 0,Y 441.105,Z 478.669,A -85,B 0,C 180,E1 -9056.107,E2 -9056.107} C_VEL
LIN {X 0,Y 440.513,Z 486.83,A -85,B 0,C 180,E1 -9059.488,E2 -9059.488} C_VEL
LIN {X 0,Y 440.055,Z 494.088,A -85,B 0,C 180,E1 -9062.409,E2 -9062.409} C_VEL
LIN {X 0,Y 439.572,Z 502.46,A -85,B 0,C 180,E1 -9065.69,E2 -9065.69} C_VEL
LIN {X 0,Y 439.202,Z 510.822,A -85,B 0,C 180,E1 -9068.897,E2 -9068.897} C_VEL
LIN {X 0,Y 438.927,Z 518.549,A -85,B 0,C 180,E1 -9071.806,E2 -9071.806} C_VEL
LIN {X 0,Y 438.786,Z 523.635,A -85,B 0,C 180,E1 -9073.7,E2 -9073.7} C_VEL
LIN {X 0,Y 440.812,Z 537.803,A -85,B 0,C 180,E1 -9074.204,E2 -9074.204} C_VEL
LIN {X 0,Y 442.026,Z 548.714,A -85,B 0,C 180,E1 -9074.732,E2 -9074.732} C_VEL
LIN {X 0,Y 441.403,Z 561.426,A -85,B 0,C 180,E1 -9075.477,E2 -9075.477} C_VEL
LIN {X 0,Y 440.834,Z 572.836,A -85,B 0,C 180,E1 -9076.339,E2 -9076.339} C_VEL
LIN {X 0,Y 440.273,Z 583.265,A -85,B 0,C 180,E1 -9077.321,E2 -9077.321} C_VEL
LIN {X 0,Y 439.701,Z 593.182,A -85,B 0,C 180,E1 -9078.475,E2 -9078.475} C_VEL
LIN {X 0,Y 439.116,Z 602.834,A -85,B 0,C 180,E1 -9079.86,E2 -9079.86} C_VEL
LIN {X 0,Y 438.81,Z 610.533,A -85,B 0,C 180,E1 -9081.248,E2 -9081.248} C_VEL
LIN {X 0,Y 438.538,Z 616.717,A -85,B 0,C 180,E1 -9082.634,E2 -9082.634} C_VEL
LIN {X 0,Y 438.396,Z 621.444,A -85,B 0,C 180,E1 -9083.965,E2 -9083.965} C_VEL
LIN {X 0,Y 438.358,Z 625.359,A -85,B 0,C 180,E1 -9085.402,E2 -9085.402} C_VEL
LIN {X 0,Y 438.332,Z 627.281,A -85,B 0,C 180,E1 -9086.323,E2 -9086.323} C_VEL
LIN {X 0,Y 438.392,Z 628.748,A -85,B 0,C 180,E1 -9087.243,E2 -9087.243} C_VEL
LIN {X 0,Y 438.366,Z 629.761,A -85,B 0,C 180,E1 -9088.163,E2 -9088.163} C_VEL
LIN {X 0,Y 438.366,Z 630.371,A -85,B 0,C 180,E1 -9089.081,E2 -9089.081} C_VEL
LIN {X 0,Y 438.337,Z 630.577,A -85,B 0,C 180,E1 -9090,E2 -9090} C_VEL
LIN {X 0,Y 438.366,Z 630.341,A -85,B 0,C 180,E1 -9090.919,E2 -9090.919} C_VEL
LIN {X 0,Y 438.368,Z 629.679,A -85,B 0,C 180,E1 -9091.837,E2 -9091.837} C_VEL
LIN {X 0,Y 438.4,Z 628.612,A -85,B 0,C 180,E1 -9092.757,E2 -9092.757} C_VEL
LIN {X 0,Y 438.342,Z 627.124,A -85,B 0,C 180,E1 -9093.677,E2 -9093.677} C_VEL
LIN {X 0,Y 438.422,Z 624.026,A -85,B 0,C 180,E1 -9095.058,E2 -9095.058} C_VEL
LIN {X 0,Y 438.448,Z 619.849,A -85,B 0,C 180,E1 -9096.442,E2 -9096.442} C_VEL
LIN {X 0,Y 438.669,Z 613.449,A -85,B 0,C 180,E1 -9098.059,E2 -9098.059} C_VEL
LIN {X 0,Y 438.956,Z 606.489,A -85,B 0,C 180,E1 -9099.446,E2 -9099.446} C_VEL
LIN {X 0,Y 439.363,Z 597.908,A -85,B 0,C 180,E1 -9100.833,E2 -9100.833} C_VEL
LIN {X 0,Y 439.921,Z 589.134,A -85,B 0,C 180,E1 -9101.987,E2 -9101.987} C_VEL
LIN {X 0,Y 440.435,Z 578.979,A -85,B 0,C 180,E1 -9103.088,E2 -9103.088} C_VEL
LIN {X 0,Y 441.086,Z 567.976,A -85,B 0,C 180,E1 -9104.063,E2 -9104.063} C_VEL
LIN {X 0,Y 441.773,Z 556.696,A -85,B 0,C 180,E1 -9104.864,E2 -9104.864} C_VEL
LIN {X 0,Y 442.098,Z 547.72,A -85,B 0,C 180,E1 -9105.384,E2 -9105.384} C_VEL
LIN {X 0,Y 440.717,Z 533.91,A -85,B 0,C 180,E1 -9106.076,E2 -9106.076} C_VEL
LIN {X 0,Y 438.767,Z 521.127,A -85,B 0,C 180,E1 -9106.593,E2 -9106.593} C_VEL
LIN {X 0,Y 438.982,Z 511.495,A -85,B 0,C 180,E1 -9110.134,E2 -9110.134} C_VEL
LIN {X 0,Y 439.247,Z 503.782,A -85,B 0,C 180,E1 -9113.079,E2 -9113.079} C_VEL
